// Device/Application/UPM03/UPMRacing_14E_StateMachine_Antigua
FUNCTION_BLOCK UPMRacing_14E_StateMachine_Antigua
VAR_INPUT
	ssMethodType: SINT;
	AMK_bSystemReady1: BOOL;
	AMK_bError1: BOOL;
	AMK_bWarn1: BOOL;
	AMK_bQuitDcOn1: BOOL;
	AMK_bQuitInverterOn1: BOOL;
	AMK_bDerating1: BOOL;
	AMK_ActualVelocity1: INT;
	AMK_TorqueCurrent1: INT;
	AMK_MagnetizingCurrent1: INT;
	AMK_TempMotor1: INT;
	AMK_TempInverter1: INT;
	AMK_ErrorInfo1: UINT;
	AMK_TempIGBT1: INT;
	AMK_bSystemReady2: BOOL;
	AMK_bError2: BOOL;
	AMK_bWarn2: BOOL;
	AMK_bQuitDcOn2: BOOL;
	AMK_bQuitInverterOn2: BOOL;
	AMK_bDerating2: BOOL;
	AMK_ActualVelocity2: INT;
	AMK_TorqueCurrent2: INT;
	AMK_MagnetizingCurrent2: INT;
	AMK_TempMotor2: INT;
	AMK_TempInverter2: INT;
	AMK_ErrorInfo2: UINT;
	AMK_TempIGBT2: INT;
	AMK_bSystemReady3: BOOL;
	AMK_bError3: BOOL;
	AMK_bWarn3: BOOL;
	AMK_bQuitDcOn3: BOOL;
	AMK_bQuitInverterOn3: BOOL;
	AMK_bDerating3: BOOL;
	AMK_ActualVelocity3: INT;
	AMK_TorqueCurrent3: INT;
	AMK_MagnetizingCurrent3: INT;
	AMK_TempMotor3: INT;
	AMK_TempInverter3: INT;
	AMK_ErrorInfo3: UINT;
	AMK_TempIGBT3: INT;
	AMK_bSystemReady4: BOOL;
	AMK_bError4: BOOL;
	AMK_bWarn4: BOOL;
	AMK_bQuitDcOn4: BOOL;
	AMK_bQuitInverterOn4: BOOL;
	AMK_bDerating4: BOOL;
	AMK_ActualVelocity4: INT;
	AMK_TorqueCurrent4: INT;
	AMK_MagnetizingCurrent4: INT;
	AMK_TempMotor4: INT;
	AMK_TempInverter4: INT;
	AMK_ErrorInfo4: UINT;
	AMK_TempIGBT4: INT;
	AccPedal_1: UINT;
	Wake_Up: UINT;
	AMK_bDcOn1_check: BOOL;
	AMK_bDcOn3_check: BOOL;
	AMK_bDcOn2_check: BOOL;
	AMK_bDcOn4_check: BOOL;
	AMK_bInverterOn1_check: BOOL;
	AMK_bInverterOn2_check: BOOL;
	AMK_bInverterOn3_check: BOOL;
	AMK_bInverterOn4_check: BOOL;
	Reset_Button: UINT;
	AccPedal_2: UINT;
	Brake_Pedal: UINT;
	Drive_Button: UINT;
	Speed: REAL;
	Shutdown_Circuit: UINT;
	BMS_Voltage: INT;
	Steering_Wheel_Angle: REAL;
	Yaw_Rate_AIM: INT;
END_VAR
VAR_OUTPUT
	AMK_bInverterOn1: BOOL;
	AMK_bDcOn1: BOOL;
	AMK_bEnable1: BOOL;
	AMK_bErrorReset1: BOOL;
	AMK_TargetVelocity1: INT;
	AMK_TorqueLimitPositiv1: INT;
	AMK_TorqueLimitNegativ1: INT;
	AMK_bInverterOn2: BOOL;
	AMK_bDcOn2: BOOL;
	AMK_bEnable2: BOOL;
	AMK_bErrorReset2: BOOL;
	AMK_TargetVelocity2: INT;
	AMK_TorqueLimitPositiv2: INT;
	AMK_TorqueLimitNegativ2: INT;
	AMK_bInverterOn3: BOOL;
	AMK_bDcOn3: BOOL;
	AMK_bEnable3: BOOL;
	AMK_bErrorReset3: BOOL;
	AMK_TargetVelocity3: INT;
	AMK_TorqueLimitPositiv3: INT;
	AMK_TorqueLimitNegativ3: INT;
	AMK_bInverterOn4: BOOL;
	AMK_bDcOn4: BOOL;
	AMK_bEnable4: BOOL;
	AMK_bErrorReset4: BOOL;
	AMK_TargetVelocity4: INT;
	AMK_TorqueLimitPositiv4: INT;
	AMK_TorqueLimitNegativ4: INT;
	Brake_Light: BOOL;
	Pre_Charge: BOOL;
	Estado: USINT;
	Inverter_Error: BOOL;
	Inverter_Warning: BOOL;
	Info_Inverter_Error: UINT;
	Estado_Error: USINT;
	Fan_Right: BOOL;
	Fan_Left: BOOL;
	RTDS_Sound: BOOL;
	AIM_TempInverter1: USINT;
	AIM_TempInverter2: USINT;
	AIM_TempInverter3: USINT;
	AIM_TempInverter4: USINT;
	AIM_TempMotor1: USINT;
	AIM_TempMotor2: USINT;
	AIM_TempMotor3: USINT;
	AIM_TempMotor4: USINT;
	Cooling_Pumps_On: BOOL;
	AIM_TorqueCurrent1: INT;
	AIM_MagnetizingCurrent1: INT;
	AIM_MagnetizingCurrent2: INT;
	AIM_MagnetizingCurrent3: INT;
	AIM_MagnetizingCurrent4: INT;
	AIM_TargetVelocity1: INT;
	AIM_TargetVelocity2: INT;
	AIM_TargetVelocity3: INT;
	AIM_TargetVelocity4: INT;
	AIM_bDerating1: BOOL;
	AIM_bDerating2: BOOL;
	AIM_bDerating3: BOOL;
	AIM_bDerating4: BOOL;
	AIM_TorqueLimitPositiv1: INT;
	AIM_TorqueLimitPositiv2: INT;
	AIM_TorqueLimitPositiv3: INT;
	AIM_TorqueLimitPositiv4: INT;
	AIM_TorqueCurrent2: INT;
	AIM_TorqueCurrent3: INT;
	AIM_TorqueCurrent4: INT;
	AIM_ActualVelocity1: INT;
	AIM_ActualVelocity2: INT;
	AIM_ActualVelocity3: INT;
	AIM_ActualVelocity4: INT;
	AIM_TempIGBT1: USINT;
	AIM_TempIGBT2: USINT;
	AIM_TempIGBT3: USINT;
	AIM_TempIGBT4: USINT;
	Throttle: REAL;
	Speed_RPM: INT;
	AIM_ErrorInfo1: UINT;
	AIM_ErrorInfo2: UINT;
	AIM_ErrorInfo3: UINT;
	AIM_ErrorInfo4: UINT;
	AIM_bError1: BOOL;
	AIM_bError2: BOOL;
	AIM_bError3: BOOL;
	AIM_bError4: BOOL;
END_VAR
VAR
	Inv_Lower_Temp: INT;
	Motor_Lower_Temp: INT;
	Braking_OffSet: UINT;
	Compare_d: BOOL;
	OutportBufferFory4: INT;
	OutportBufferFory3: INT;
	OutportBufferFory2: INT;
	x_l: INT;
	AMK_bError4_g: BOOL;
	AMK_bError3_n: BOOL;
	AMK_bError2_e: BOOL;
	AMK_bError1_k: BOOL;
	AMK_ErrorInfo4_oa: UINT;
	AMK_ErrorInfo3_p: UINT;
	AMK_ErrorInfo2_a: UINT;
	AMK_ErrorInfo1_h: UINT;
	AMK_MagnetizingCurrent4_m: INT;
	AMK_MagnetizingCurrent3_f: INT;
	AMK_MagnetizingCurrent2_a: INT;
	AMK_MagnetizingCurrent1_j: INT;
	AMK_ActualVelocity4_c: INT;
	AMK_ActualVelocity3_i: INT;
	AMK_ActualVelocity2_e: INT;
	AMK_ActualVelocity1_l: INT;
	AMK_TorqueLimitPositiv4_l: INT;
	AMK_TorqueLimitPositiv3_m: INT;
	AMK_TorqueLimitPositiv2_o: INT;
	AMK_TorqueLimitPositiv1_e: INT;
	AMK_TargetVelocity4_p: INT;
	AMK_TargetVelocity3_h: INT;
	AMK_TargetVelocity2_c: INT;
	AMK_TargetVelocity1_gb: INT;
	AMK_TorqueCurrent4_b: INT;
	AMK_TorqueCurrent3_p: INT;
	AMK_TorqueCurrent2_b: INT;
	AMK_TorqueCurrent1_m: INT;
	AMK_bDerating4_p: BOOL;
	AMK_bDerating3_g: BOOL;
	AMK_bDerating2_p: BOOL;
	AMK_bDerating1_h: BOOL;
	DataTypeConversion3_o: USINT;
	DataTypeConversion1_n: USINT;
	DataTypeConversion2_m: USINT;
	DataTypeConversion_b: USINT;
	DataTypeConversion3_p: USINT;
	DataTypeConversion1_g: USINT;
	DataTypeConversion2_e: USINT;
	DataTypeConversion_e: USINT;
	DataTypeConversion3_e: USINT;
	DataTypeConversion1_c: USINT;
	DataTypeConversion2_f: USINT;
	DataTypeConversion_h: USINT;
	b_Add: UINT;
	OutportBufferForAMK_bErrorReset4: BOOL;
	OutportBufferForAMK_bErrorReset3: BOOL;
	OutportBufferForAMK_bErrorReset2: BOOL;
	Compare: BOOL;
	LogicalOperator1: BOOL;
	LogicalOperator: BOOL;
	Saturation: REAL;
	OutportBufferForAMK_TargetVelocity4: INT;
	OutportBufferForAMK_TargetVelocity3: INT;
	OutportBufferForAMK_TargetVelocity2: INT;
	DataTypeConversion3: INT;
	OutportBufferForAMK_TorqueLimitNegativ4: INT;
	OutportBufferForAMK_TorqueLimitNegativ3: INT;
	OutportBufferForAMK_TorqueLimitNegativ2: INT;
	DataTypeConversion6: INT;
	DataTypeConversion: INT;
	DataTypeConversion5: INT;
	DataTypeConversion4: INT;
	DataTypeConversion2: INT;
	DataTypeConversion1: INT;
	is_active_c3_UPMRacing_14E_StateMachine: USINT;
	is_CAR: USINT;
	is_SHUTDOWN_SEQUENCE: USINT;
	temporalCounter_i1: PLC_CODER_TIMER;
	Cooling_Enable: BOOL;
	x: INT;
	is_IDLE: USINT;
	is_DRIVE: USINT;
	BMS_Voltage_Min: INT;
	b_AccPedal_2: UINT;
	b_AccPedal_1: UINT;
	b_Yaw_Rate_AIM: INT;
	b_Steering_Wheel_Angle: REAL;
	Throttle_a: REAL;
	b_AMK_ActualVelocity4: INT;
	b_AMK_ActualVelocity3: INT;
	b_AMK_ActualVelocity2: INT;
	b_AMK_ActualVelocity1: INT;
	is_POWER_MOTOR_ON: USINT;
	is_ERROR_INVERTER: USINT;
	b_AMK_bWarn4: BOOL;
	b_AMK_bWarn3: BOOL;
	b_AMK_bWarn2: BOOL;
	b_AMK_bWarn1: BOOL;
	b_AMK_bError4: BOOL;
	b_AMK_bError3: BOOL;
	b_AMK_bError2: BOOL;
	b_AMK_bError1: BOOL;
	AMK_bError4_a: BOOL;
	AMK_bError3_d: BOOL;
	AMK_bError2_h: BOOL;
	AMK_bError1_b: BOOL;
	b_AMK_ErrorInfo4: UINT;
	b_AMK_ErrorInfo3: UINT;
	b_AMK_ErrorInfo2: UINT;
	b_AMK_ErrorInfo1: UINT;
	is_BRAKE_LIGHT: USINT;
	is_COOLING_RIGHT: USINT;
	Fan_Upper_Speed: UINT;
	Motor_Upper_Temp: INT;
	Fan_Lower_Speed: UINT;
	is_COOLING_LEFT: USINT;
	b_AMK_TempInverter4: INT;
	b_AMK_TempInverter3: INT;
	b_AMK_TempInverter2: INT;
	b_AMK_TempInverter1: INT;
	b_AMK_TempMotor4: INT;
	b_AMK_TempMotor3: INT;
	b_AMK_TempMotor2: INT;
	b_AMK_TempMotor1: INT;
	b_AMK_TempIGBT4: INT;
	b_AMK_TempIGBT3: INT;
	b_AMK_TempIGBT2: INT;
	b_AMK_TempIGBT1: INT;
	b_AMK_bDerating4: BOOL;
	b_AMK_bDerating3: BOOL;
	b_AMK_bDerating2: BOOL;
	b_AMK_bDerating1: BOOL;
	b_AMK_TorqueCurrent4: INT;
	b_AMK_TorqueCurrent3: INT;
	b_AMK_TorqueCurrent2: INT;
	b_AMK_TorqueCurrent1: INT;
	AMK_TargetVelocity4_b: INT;
	AMK_TargetVelocity3_m: INT;
	AMK_TargetVelocity2_m: INT;
	AMK_TargetVelocity1_g: INT;
	AMK_TorqueLimitPositiv4_h: INT;
	AMK_TorqueLimitPositiv3_i: INT;
	AMK_TorqueLimitPositiv2_l: INT;
	AMK_TorqueLimitPositiv1_c: INT;
	AMK_ActualVelocity4_k: INT;
	AMK_ActualVelocity3_f: INT;
	AMK_ActualVelocity2_n: INT;
	AMK_ActualVelocity1_b: INT;
	b_AMK_MagnetizingCurrent4: INT;
	b_AMK_MagnetizingCurrent3: INT;
	b_AMK_MagnetizingCurrent2: INT;
	b_AMK_MagnetizingCurrent1: INT;
	AMK_bError4_p: BOOL;
	AMK_bError3_p: BOOL;
	AMK_bError2_g: BOOL;
	AMK_bError1_d: BOOL;
	AMK_ErrorInfo4_o: UINT;
	AMK_ErrorInfo3_l: UINT;
	AMK_ErrorInfo2_f: UINT;
	AMK_ErrorInfo1_n: UINT;
	Inv_Upper_Temp: INT;
	i0_b_Constant: b_Constant;
	i0_Throttle_Control: Throttle_Control;
	i0_Yaw_Control: Yaw_Control;
	i0_Error_Control: Error_Control;
	i0_Error_RESET: Error_RESET;
	i0_Error_Info: Error_Info;
	i0_Temp_Inverter: Temp_Inverter;
	i0_Temp_Motor: Temp_Motor;
	i0_Temp_IGBT: Temp_IGBT;
	i0_Derating: Derating;
	i0_TorqueCurrent: TorqueCurrent;
	i0_TargetVelocity: TargetVelocity;
	i0_TorqueLimitPositiv: TorqueLimitPositiv;
	i0_ActualVelocity: ActualVelocity;
	i0_MagnetizingCurrent: MagnetizingCurrent;
	i0_ErrorInfo: ErrorInfo;
	sf_internal_predicateOutput: BOOL;
	tmp: UINT;
	temp1: UINT;
	temp2: UINT;
	temp3: USINT;
	temp4: USINT;
	temp5: USINT;
	temp6: USINT;
	temp7: UINT;
	temp8: BOOL;
	temp9: BOOL;
	temp10: BOOL;
	temp11: REAL;
	temp12: INT;
	temp13: INT;
	temp14: INT;
	temp15: INT;
	temp16: INT;
	temp17: INT;
	temp18: INT;
	temp19: INT;
	temp20: INT;
	temp21: INT;
	temp22: INT;
	temp23: INT;
	temp24: INT;
	
	//Llamadas a las funciones de CAN (Copiar)
	
	CAN_RX_V_1_2:CAN_RX_V_1_2;
	CAN_RX_Inverters:CAN_RX_Inverters;
	
	CAN_TX_V_1_4:CAN_TX_V_1_4;
	CAN_TX_Inverters:CAN_TX_Inverters;
	
END_VAR


CAN_RX_V_1_2( 
	    		
		(*DATA LOGGER*) (*
			DL_Msg_Cntr_CAN => DL_Msg_Cntr,
			DL_Status_CAN => DL_Status,
			DL_Power_CAN => DL_Power,
			DL_Voltage_CAN => DL_Voltage,
			DL_Current_CAN => DL_Current,
		(*FIN DATA LOGGER*) *)
		
		(*BMS*)
			BatVoltage_MSB_CAN => BMS_Voltage,
		(*__*)
		
		(*AIM RX*) 
			Speed_CAN => Speed,
			//AIM_Long_Acc_CAN => Long_Acc,
			//AIM_Lat_Acc_CAN => Lat_Acc,
			Yaw_Rate_AIM_CAN => Yaw_Rate_AIM, 
			
			Steering_Wheel_Angle_CAN => Steering_Wheel_Angle,
		(*__*)
		
			); 	
(*_________*)		
		
CAN_RX_Inverters( 
	
		(*INVERTERS*)
		AMK_bSystemReady1_CAN=>AMK_bSystemReady1,
		AMK_bError1_CAN=>AMK_bError1,
		AMK_bWarn1_CAN=>AMK_bWarn1,
		AMK_bQuitDcOn1_CAN=>AMK_bQuitDcOn1,
		AMK_bDcOn1_check_CAN=>AMK_bDcOn1_check,
		AMK_bQuitInverterOn1_CAN=>AMK_bQuitInverterOn1,
		AMK_bInverterOn1_check_CAN=>AMK_bInverterOn1_check,
		AMK_bDerating1_CAN=>AMK_bDerating1,
		AMK_ActualVelocity1_CAN=>AMK_ActualVelocity1,
		AMK_TorqueCurrent1_CAN=>AMK_TorqueCurrent1,
		AMK_MagnetizingCurrent1_CAN=>AMK_MagnetizingCurrent1,
		AMK_TempMotor1_CAN=>AMK_TempMotor1,
		AMK_TempInverter1_CAN=>AMK_TempInverter1,
		AMK_ErrorInfo1_CAN=>AMK_ErrorInfo1,
		AMK_TempIGBT1_CAN=>AMK_TempIGBT1,
		
		
		AMK_bSystemReady2_CAN=>AMK_bSystemReady2,
		AMK_bError2_CAN=>AMK_bError2,
		AMK_bWarn2_CAN=>AMK_bWarn2,
		AMK_bQuitDcOn2_CAN=>AMK_bQuitDcOn2,
		AMK_bDcOn2_check_CAN=>AMK_bDcOn2_check,
		AMK_bQuitInverterOn2_CAN=>AMK_bQuitInverterOn2,
		AMK_bInverterOn2_check_CAN=>AMK_bInverterOn2_check,
		AMK_bDerating2_CAN=>AMK_bDerating2,
		AMK_ActualVelocity2_CAN=>AMK_ActualVelocity2,
		AMK_TorqueCurrent2_CAN=>AMK_TorqueCurrent2,
		AMK_MagnetizingCurrent2_CAN=>AMK_MagnetizingCurrent2,
		AMK_TempMotor2_CAN=>AMK_TempMotor2,
		AMK_TempInverter2_CAN=>AMK_TempInverter2,
		AMK_ErrorInfo2_CAN=>AMK_ErrorInfo2,
		AMK_TempIGBT2_CAN=>AMK_TempIGBT2,
		
		
		AMK_bSystemReady3_CAN=>AMK_bSystemReady3,
		AMK_bError3_CAN=>AMK_bError3,
		AMK_bWarn3_CAN=>AMK_bWarn3,
		AMK_bQuitDcOn3_CAN=>AMK_bQuitDcOn3,
		AMK_bDcOn3_check_CAN=>AMK_bDcOn3_check,
		AMK_bQuitInverterOn3_CAN=>AMK_bQuitInverterOn3,
		AMK_bInverterOn3_check_CAN=>AMK_bInverterOn3_check,
		AMK_bDerating3_CAN=>AMK_bDerating3,
		AMK_ActualVelocity3_CAN=>AMK_ActualVelocity3,
		AMK_TorqueCurrent3_CAN=>AMK_TorqueCurrent3,
		AMK_MagnetizingCurrent3_CAN=>AMK_MagnetizingCurrent3,
		AMK_TempMotor3_CAN=>AMK_TempMotor3,
		AMK_TempInverter3_CAN=>AMK_TempInverter3,
		AMK_ErrorInfo3_CAN=>AMK_ErrorInfo3,
		AMK_TempIGBT3_CAN=>AMK_TempIGBT3,
		
		
		AMK_bSystemReady4_CAN=>AMK_bSystemReady4,
		AMK_bError4_CAN=>AMK_bError4,
		AMK_bWarn4_CAN=>AMK_bWarn4,
		AMK_bQuitDcOn4_CAN=>AMK_bQuitDcOn4,
		AMK_bDcOn4_check_CAN=>AMK_bDcOn4_check,
		AMK_bQuitInverterOn4_CAN=>AMK_bQuitInverterOn4,
		AMK_bInverterOn4_check_CAN=>AMK_bInverterOn4_check,
		AMK_bDerating4_CAN=>AMK_bDerating4,
		AMK_ActualVelocity4_CAN=>AMK_ActualVelocity4,
		AMK_TorqueCurrent4_CAN=>AMK_TorqueCurrent4,
		AMK_MagnetizingCurrent4_CAN=>AMK_MagnetizingCurrent4,
		AMK_TempMotor4_CAN=>AMK_TempMotor4,
		AMK_TempInverter4_CAN=>AMK_TempInverter4,
		AMK_ErrorInfo4_CAN=>AMK_ErrorInfo4,
		AMK_TempIGBT4_CAN=>AMK_TempIGBT4
		
		);

(*___________________*)

CASE ssMethodType OF
    SS_INITIALIZE: 
        (* SystemInitialize for Chart: '<Root>/UPMRacing_14E_StateMachine' incorporates:
         *  Outport: '<Root>/AIM_ErrorInfo1'
         *  Outport: '<Root>/AIM_ErrorInfo2'
         *  Outport: '<Root>/AIM_ErrorInfo3'
         *  Outport: '<Root>/AIM_ErrorInfo4'
         *  Outport: '<Root>/AIM_TargetVelocity1'
         *  Outport: '<Root>/AIM_TargetVelocity2'
         *  Outport: '<Root>/AIM_TargetVelocity3'
         *  Outport: '<Root>/AIM_TargetVelocity4'
         *  Outport: '<Root>/AIM_TorqueLimitPositiv1'
         *  Outport: '<Root>/AIM_TorqueLimitPositiv2'
         *  Outport: '<Root>/AIM_TorqueLimitPositiv3'
         *  Outport: '<Root>/AIM_TorqueLimitPositiv4'
         *  Outport: '<Root>/AIM_bError1'
         *  Outport: '<Root>/AIM_bError2'
         *  Outport: '<Root>/AIM_bError3'
         *  Outport: '<Root>/AIM_bError4'
         *  Outport: '<Root>/AMK_TargetVelocity1'
         *  Outport: '<Root>/AMK_TargetVelocity2'
         *  Outport: '<Root>/AMK_TargetVelocity3'
         *  Outport: '<Root>/AMK_TargetVelocity4'
         *  Outport: '<Root>/AMK_TorqueLimitNegativ1'
         *  Outport: '<Root>/AMK_TorqueLimitNegativ2'
         *  Outport: '<Root>/AMK_TorqueLimitNegativ3'
         *  Outport: '<Root>/AMK_TorqueLimitNegativ4'
         *  Outport: '<Root>/AMK_TorqueLimitPositiv1'
         *  Outport: '<Root>/AMK_TorqueLimitPositiv2'
         *  Outport: '<Root>/AMK_TorqueLimitPositiv3'
         *  Outport: '<Root>/AMK_TorqueLimitPositiv4'
         *  Outport: '<Root>/AMK_bDcOn1'
         *  Outport: '<Root>/AMK_bDcOn2'
         *  Outport: '<Root>/AMK_bDcOn3'
         *  Outport: '<Root>/AMK_bDcOn4'
         *  Outport: '<Root>/AMK_bEnable1'
         *  Outport: '<Root>/AMK_bEnable2'
         *  Outport: '<Root>/AMK_bEnable3'
         *  Outport: '<Root>/AMK_bEnable4'
         *  Outport: '<Root>/AMK_bErrorReset1'
         *  Outport: '<Root>/AMK_bErrorReset2'
         *  Outport: '<Root>/AMK_bErrorReset3'
         *  Outport: '<Root>/AMK_bErrorReset4'
         *  Outport: '<Root>/AMK_bInverterOn1'
         *  Outport: '<Root>/AMK_bInverterOn2'
         *  Outport: '<Root>/AMK_bInverterOn3'
         *  Outport: '<Root>/AMK_bInverterOn4'
         *  Outport: '<Root>/Fan_Left'
         *  Outport: '<Root>/Fan_Right'
         *  Outport: '<Root>/RTDS_Sound'
         *  Outport: '<Root>/Speed_RPM' *)
        is_BRAKE_LIGHT := UPMRacing_14E_StateMachine_IN_NO_ACTIVE_CHILD;
        is_CAR := UPMRacing_14E_StateMachine_IN_NO_ACTIVE_CHILD;
        is_DRIVE := UPMRacing_14E_StateMachine_IN_NO_ACTIVE_CHILD;
        temporalCounter_i1(timerAction := 1, maxTime := 0);
        is_IDLE := UPMRacing_14E_StateMachine_IN_NO_ACTIVE_CHILD;
        is_POWER_MOTOR_ON := UPMRacing_14E_StateMachine_IN_NO_ACTIVE_CHILD;
        temporalCounter_i1(timerAction := 1, maxTime := 0);
        is_SHUTDOWN_SEQUENCE := UPMRacing_14E_StateMachine_IN_NO_ACTIVE_CHILD;
        temporalCounter_i1(timerAction := 1, maxTime := 0);
        is_COOLING_LEFT := UPMRacing_14E_StateMachine_IN_NO_ACTIVE_CHILD;
        is_COOLING_RIGHT := UPMRacing_14E_StateMachine_IN_NO_ACTIVE_CHILD;
        is_ERROR_INVERTER := UPMRacing_14E_StateMachine_IN_NO_ACTIVE_CHILD;
        is_active_c3_UPMRacing_14E_StateMachine := 0;
        Braking_OffSet := 3850;
        Motor_Upper_Temp := 700;
        Motor_Lower_Temp := 500;
        Fan_Upper_Speed := 350;
        Fan_Lower_Speed := 350;
        Inv_Lower_Temp := 250;
        Inv_Upper_Temp := 300;
        Cooling_Enable := FALSE;
        BMS_Voltage_Min := 306;
        AMK_bInverterOn1 := FALSE;
        AMK_bDcOn1 := FALSE;
        AMK_bEnable1 := FALSE;
        AMK_bErrorReset1 := FALSE;
        AMK_TargetVelocity1 := 0;
        AMK_TorqueLimitPositiv1 := 0;
        AMK_TorqueLimitNegativ1 := 0;
        AMK_bInverterOn2 := FALSE;
        AMK_bDcOn2 := FALSE;
        AMK_bEnable2 := FALSE;
        AMK_bErrorReset2 := FALSE;
        AMK_TargetVelocity2 := 0;
        AMK_TorqueLimitPositiv2 := 0;
        AMK_TorqueLimitNegativ2 := 0;
        AMK_bInverterOn3 := FALSE;
        AMK_bDcOn3 := FALSE;
        AMK_bEnable3 := FALSE;
        AMK_bErrorReset3 := FALSE;
        AMK_TargetVelocity3 := 0;
        AMK_TorqueLimitPositiv3 := 0;
        AMK_TorqueLimitNegativ3 := 0;
        AMK_bInverterOn4 := FALSE;
        AMK_bDcOn4 := FALSE;
        AMK_bEnable4 := FALSE;
        AMK_bErrorReset4 := FALSE;
        AMK_TargetVelocity4 := 0;
        AMK_TorqueLimitPositiv4 := 0;
        AMK_TorqueLimitNegativ4 := 0;
        Fan_Right := FALSE;
        Fan_Left := FALSE;
        RTDS_Sound := FALSE;
        AIM_TargetVelocity1 := 0;
        AIM_TargetVelocity2 := 0;
        AIM_TargetVelocity3 := 0;
        AIM_TargetVelocity4 := 0;
        AIM_TorqueLimitPositiv1 := 0;
        AIM_TorqueLimitPositiv2 := 0;
        AIM_TorqueLimitPositiv3 := 0;
        AIM_TorqueLimitPositiv4 := 0;
        Speed_RPM := 0;
        AIM_ErrorInfo1 := 0;
        AIM_ErrorInfo2 := 0;
        AIM_ErrorInfo3 := 0;
        AIM_ErrorInfo4 := 0;
        AIM_bError1 := FALSE;
        AIM_bError2 := FALSE;
        AIM_bError3 := FALSE;
        AIM_bError4 := FALSE;
        i0_Yaw_Control(ssMethodType := SS_INITIALIZE, AMK_ActualVelocity1 := b_AMK_ActualVelocity1, AMK_ActualVelocity2 := b_AMK_ActualVelocity2, AMK_ActualVelocity3 := b_AMK_ActualVelocity3, AMK_ActualVelocity4 := b_AMK_ActualVelocity4, Throttle := Throttle_a, Steering_Wheel_Angle := b_Steering_Wheel_Angle, Yaw_Rate_AIM := b_Yaw_Rate_AIM);
        OutportBufferForAMK_TargetVelocity4 := temp24;
        OutportBufferForAMK_TargetVelocity3 := temp23;
        OutportBufferForAMK_TargetVelocity2 := temp22;
        DataTypeConversion3 := temp21;
        OutportBufferForAMK_TorqueLimitNegativ4 := temp20;
        OutportBufferForAMK_TorqueLimitNegativ3 := temp19;
        OutportBufferForAMK_TorqueLimitNegativ2 := temp18;
        DataTypeConversion6 := temp17;
        DataTypeConversion := temp16;
        DataTypeConversion5 := temp15;
        DataTypeConversion4 := temp14;
        DataTypeConversion2 := temp13;
        DataTypeConversion1 := temp12;
        i0_b_Constant(ssMethodType := SS_INITIALIZE, x := x);
        OutportBufferFory4 := temp15;
        OutportBufferFory3 := temp14;
        OutportBufferFory2 := temp13;
        x_l := temp12;
        i0_Throttle_Control(ssMethodType := SS_INITIALIZE, AccPedal_1 := b_AccPedal_1, AccPedal_2 := b_AccPedal_2,  Brake_Light2 := Brake_Pedal);
        Compare_d := sf_internal_predicateOutput;
        Saturation := temp11;
        i0_Error_Control(ssMethodType := SS_INITIALIZE, AMK_bError1 := b_AMK_bError1, AMK_bError2 := b_AMK_bError2, AMK_bError3 := b_AMK_bError3, AMK_bError4 := b_AMK_bError4, AMK_bWarn1 := b_AMK_bWarn1, AMK_bWarn2 := b_AMK_bWarn2, AMK_bWarn3 := b_AMK_bWarn3, AMK_bWarn4 := b_AMK_bWarn4);
        LogicalOperator1 := temp10;
        LogicalOperator := sf_internal_predicateOutput;
        i0_Error_RESET(ssMethodType := SS_INITIALIZE);
        OutportBufferForAMK_bErrorReset4 := temp9;
        OutportBufferForAMK_bErrorReset3 := temp8;
        OutportBufferForAMK_bErrorReset2 := temp10;
        Compare := sf_internal_predicateOutput;
        i0_Error_Info(ssMethodType := SS_INITIALIZE, AMK_ErrorInfo1 := b_AMK_ErrorInfo1, AMK_ErrorInfo2 := b_AMK_ErrorInfo2, AMK_ErrorInfo3 := b_AMK_ErrorInfo3, AMK_ErrorInfo4 := b_AMK_ErrorInfo4, AMK_bError1 := AMK_bError1_b, AMK_bError2 := AMK_bError2_h, AMK_bError3 := AMK_bError3_d, AMK_bError4 := AMK_bError4_a);
        b_Add := temp7;
        i0_Temp_Inverter(ssMethodType := SS_INITIALIZE, AMK_TempInverter1 := b_AMK_TempInverter1, AMK_TempInverter2 := b_AMK_TempInverter2, AMK_TempInverter3 := b_AMK_TempInverter3, AMK_TempInverter4 := b_AMK_TempInverter4);
        DataTypeConversion3_e := temp6;
        DataTypeConversion1_c := temp5;
        DataTypeConversion2_f := temp4;
        DataTypeConversion_h := temp3;
        i0_Temp_Motor(ssMethodType := SS_INITIALIZE, AMK_TempMotor1 := b_AMK_TempMotor1, AMK_TempMotor2 := b_AMK_TempMotor2, AMK_TempMotor3 := b_AMK_TempMotor3, AMK_TempMotor4 := b_AMK_TempMotor4);
        DataTypeConversion3_p := temp6;
        DataTypeConversion1_g := temp5;
        DataTypeConversion2_e := temp4;
        DataTypeConversion_e := temp3;
        i0_Temp_IGBT(ssMethodType := SS_INITIALIZE, AMK_TempIGBT1 := b_AMK_TempIGBT1, AMK_TempIGBT2 := b_AMK_TempIGBT2, AMK_TempIGBT3 := b_AMK_TempIGBT3, AMK_TempIGBT4 := b_AMK_TempIGBT4);
        DataTypeConversion3_o := temp6;
        DataTypeConversion1_n := temp5;
        DataTypeConversion2_m := temp4;
        DataTypeConversion_b := temp3;
        i0_Derating(ssMethodType := SS_INITIALIZE, AMK_bDerating1 := b_AMK_bDerating1, AMK_bDerating2 := b_AMK_bDerating2, AMK_bDerating3 := b_AMK_bDerating3, AMK_bDerating4 := b_AMK_bDerating4);
        AMK_bDerating4_p := temp9;
        AMK_bDerating3_g := temp8;
        AMK_bDerating2_p := temp10;
        AMK_bDerating1_h := sf_internal_predicateOutput;
        i0_MagnetizingCurrent(ssMethodType := SS_INITIALIZE, AMK_MagnetizingCurrent1 := b_AMK_MagnetizingCurrent1, AMK_MagnetizingCurrent2 := b_AMK_MagnetizingCurrent2, AMK_MagnetizingCurrent3 := b_AMK_MagnetizingCurrent3, AMK_MagnetizingCurrent4 := b_AMK_MagnetizingCurrent4);
        AMK_MagnetizingCurrent4_m := temp15;
        AMK_MagnetizingCurrent3_f := temp14;
        AMK_MagnetizingCurrent2_a := temp13;
        AMK_MagnetizingCurrent1_j := temp12;
        i0_TorqueCurrent(ssMethodType := SS_INITIALIZE, AMK_TorqueCurrent1 := b_AMK_TorqueCurrent1, AMK_TorqueCurrent2 := b_AMK_TorqueCurrent2, AMK_TorqueCurrent3 := b_AMK_TorqueCurrent3, AMK_TorqueCurrent4 := b_AMK_TorqueCurrent4);
        AMK_TorqueCurrent4_b := temp15;
        AMK_TorqueCurrent3_p := temp14;
        AMK_TorqueCurrent2_b := temp13;
        AMK_TorqueCurrent1_m := temp12;
        i0_TargetVelocity(ssMethodType := SS_INITIALIZE, AMK_TargetVelocity1 := AMK_TargetVelocity1_g, AMK_TargetVelocity2 := AMK_TargetVelocity2_m, AMK_TargetVelocity3 := AMK_TargetVelocity3_m, AMK_TargetVelocity4 := AMK_TargetVelocity4_b);
        AMK_TargetVelocity4_p := temp15;
        AMK_TargetVelocity3_h := temp14;
        AMK_TargetVelocity2_c := temp13;
        AMK_TargetVelocity1_gb := temp12;
        i0_TorqueLimitPositiv(ssMethodType := SS_INITIALIZE, AMK_TorqueLimitPositiv1 := AMK_TorqueLimitPositiv1_c, AMK_TorqueLimitPositiv2 := AMK_TorqueLimitPositiv2_l, AMK_TorqueLimitPositiv3 := AMK_TorqueLimitPositiv3_i, AMK_TorqueLimitPositiv4 := AMK_TorqueLimitPositiv4_h);
        AMK_TorqueLimitPositiv4_l := temp15;
        AMK_TorqueLimitPositiv3_m := temp14;
        AMK_TorqueLimitPositiv2_o := temp13;
        AMK_TorqueLimitPositiv1_e := temp12;
        i0_ActualVelocity(ssMethodType := SS_INITIALIZE, AMK_ActualVelocity1 := AMK_ActualVelocity1_b, AMK_ActualVelocity2 := AMK_ActualVelocity2_n, AMK_ActualVelocity3 := AMK_ActualVelocity3_f, AMK_ActualVelocity4 := AMK_ActualVelocity4_k);
        AMK_ActualVelocity4_c := temp15;
        AMK_ActualVelocity3_i := temp14;
        AMK_ActualVelocity2_e := temp13;
        AMK_ActualVelocity1_l := temp12;
        i0_ErrorInfo(ssMethodType := SS_INITIALIZE, AMK_ErrorInfo1 := AMK_ErrorInfo1_n, AMK_ErrorInfo2 := AMK_ErrorInfo2_f, AMK_ErrorInfo3 := AMK_ErrorInfo3_l, AMK_ErrorInfo4 := AMK_ErrorInfo4_o, AMK_bError1 := AMK_bError1_d, AMK_bError2 := AMK_bError2_g, AMK_bError3 := AMK_bError3_p, AMK_bError4 := AMK_bError4_p);
        AMK_bError4_g := temp9;
        AMK_bError3_n := temp8;
        AMK_bError2_e := temp10;
        AMK_bError1_k := sf_internal_predicateOutput;
        AMK_ErrorInfo4_oa := temp2;
        AMK_ErrorInfo3_p := temp1;
        AMK_ErrorInfo2_a := tmp;
        AMK_ErrorInfo1_h := temp7;
    SS_STEP: 
        (* Chart: '<Root>/UPMRacing_14E_StateMachine' incorporates:
         *  Outport: '<Root>/AIM_ActualVelocity1'
         *  Outport: '<Root>/AIM_ActualVelocity2'
         *  Outport: '<Root>/AIM_ActualVelocity3'
         *  Outport: '<Root>/AIM_ActualVelocity4'
         *  Outport: '<Root>/AIM_ErrorInfo1'
         *  Outport: '<Root>/AIM_ErrorInfo2'
         *  Outport: '<Root>/AIM_ErrorInfo3'
         *  Outport: '<Root>/AIM_ErrorInfo4'
         *  Outport: '<Root>/AIM_MagnetizingCurrent1'
         *  Outport: '<Root>/AIM_MagnetizingCurrent2'
         *  Outport: '<Root>/AIM_MagnetizingCurrent3'
         *  Outport: '<Root>/AIM_MagnetizingCurrent4'
         *  Outport: '<Root>/AIM_TargetVelocity1'
         *  Outport: '<Root>/AIM_TargetVelocity2'
         *  Outport: '<Root>/AIM_TargetVelocity3'
         *  Outport: '<Root>/AIM_TargetVelocity4'
         *  Outport: '<Root>/AIM_TempIGBT1'
         *  Outport: '<Root>/AIM_TempIGBT2'
         *  Outport: '<Root>/AIM_TempIGBT3'
         *  Outport: '<Root>/AIM_TempIGBT4'
         *  Outport: '<Root>/AIM_TempInverter1'
         *  Outport: '<Root>/AIM_TempInverter2'
         *  Outport: '<Root>/AIM_TempInverter3'
         *  Outport: '<Root>/AIM_TempInverter4'
         *  Outport: '<Root>/AIM_TempMotor1'
         *  Outport: '<Root>/AIM_TempMotor2'
         *  Outport: '<Root>/AIM_TempMotor3'
         *  Outport: '<Root>/AIM_TempMotor4'
         *  Outport: '<Root>/AIM_TorqueCurrent1'
         *  Outport: '<Root>/AIM_TorqueCurrent2'
         *  Outport: '<Root>/AIM_TorqueCurrent3'
         *  Outport: '<Root>/AIM_TorqueCurrent4'
         *  Outport: '<Root>/AIM_TorqueLimitPositiv1'
         *  Outport: '<Root>/AIM_TorqueLimitPositiv2'
         *  Outport: '<Root>/AIM_TorqueLimitPositiv3'
         *  Outport: '<Root>/AIM_TorqueLimitPositiv4'
         *  Outport: '<Root>/AIM_bDerating1'
         *  Outport: '<Root>/AIM_bDerating2'
         *  Outport: '<Root>/AIM_bDerating3'
         *  Outport: '<Root>/AIM_bDerating4'
         *  Outport: '<Root>/AIM_bError1'
         *  Outport: '<Root>/AIM_bError2'
         *  Outport: '<Root>/AIM_bError3'
         *  Outport: '<Root>/AIM_bError4'
         *  Outport: '<Root>/AMK_TargetVelocity1'
         *  Outport: '<Root>/AMK_TargetVelocity2'
         *  Outport: '<Root>/AMK_TargetVelocity3'
         *  Outport: '<Root>/AMK_TargetVelocity4'
         *  Outport: '<Root>/AMK_TorqueLimitNegativ1'
         *  Outport: '<Root>/AMK_TorqueLimitNegativ2'
         *  Outport: '<Root>/AMK_TorqueLimitNegativ3'
         *  Outport: '<Root>/AMK_TorqueLimitNegativ4'
         *  Outport: '<Root>/AMK_TorqueLimitPositiv1'
         *  Outport: '<Root>/AMK_TorqueLimitPositiv2'
         *  Outport: '<Root>/AMK_TorqueLimitPositiv3'
         *  Outport: '<Root>/AMK_TorqueLimitPositiv4'
         *  Outport: '<Root>/AMK_bDcOn1'
         *  Outport: '<Root>/AMK_bDcOn2'
         *  Outport: '<Root>/AMK_bDcOn3'
         *  Outport: '<Root>/AMK_bDcOn4'
         *  Outport: '<Root>/AMK_bEnable1'
         *  Outport: '<Root>/AMK_bEnable2'
         *  Outport: '<Root>/AMK_bEnable3'
         *  Outport: '<Root>/AMK_bEnable4'
         *  Outport: '<Root>/AMK_bErrorReset1'
         *  Outport: '<Root>/AMK_bErrorReset2'
         *  Outport: '<Root>/AMK_bErrorReset3'
         *  Outport: '<Root>/AMK_bErrorReset4'
         *  Outport: '<Root>/AMK_bInverterOn1'
         *  Outport: '<Root>/AMK_bInverterOn2'
         *  Outport: '<Root>/AMK_bInverterOn3'
         *  Outport: '<Root>/AMK_bInverterOn4'
         *  Outport: '<Root>/Brake_Light'
         *  Outport: '<Root>/Cooling_Pumps_On'
         *  Outport: '<Root>/Estado'
         *  Outport: '<Root>/Fan_Left'
         *  Outport: '<Root>/Fan_Right'
         *  Outport: '<Root>/Info_Inverter_Error'
         *  Outport: '<Root>/Inverter_Error'
         *  Outport: '<Root>/Inverter_Warning'
         *  Outport: '<Root>/Pre_Charge'
         *  Outport: '<Root>/RTDS_Sound'
         *  Outport: '<Root>/Speed_RPM'
         *  Outport: '<Root>/Throttle' *)
        (* Gateway: UPMRacing_14E_StateMachine *)
        (* During: UPMRacing_14E_StateMachine *)

        IF is_active_c3_UPMRacing_14E_StateMachine = 0 THEN 
            (* Entry: UPMRacing_14E_StateMachine *)
            is_active_c3_UPMRacing_14E_StateMachine := 1;
            (* Entry Internal: UPMRacing_14E_StateMachine *)
            (* Entry Internal 'CAR': '<S1>:380' *)
            (* Transition: '<S1>:138' *)
            is_CAR := UPMRacing_14E_StateMachine_IN_IDLE;
            (* Entry 'IDLE': '<S1>:333' *)
            (* '<S1>:333:3' Cooling_Enable = false; *)
            Cooling_Enable := FALSE;
            (* '<S1>:333:4' [AMK_TargetVelocity1, AMK_TargetVelocity2, AMK_TargetVelocity3, AMK_TargetVelocity4... *)
            (* '<S1>:333:5'      ]=Constant(int16(0)); *)
            (* Simulink Function 'Constant': '<S1>:190' *)
            x := 0;
            i0_b_Constant(ssMethodType := SS_OUTPUT, x := x);
            temp12 := i0_b_Constant.y1;
            temp13 := i0_b_Constant.y2;
            temp14 := i0_b_Constant.y3;
            temp15 := i0_b_Constant.y4;
            OutportBufferFory4 := temp15;
            OutportBufferFory3 := temp14;
            OutportBufferFory2 := temp13;
            x_l := temp12;
            AMK_TargetVelocity1 := x_l;
            AMK_TargetVelocity2 := OutportBufferFory2;
            AMK_TargetVelocity3 := OutportBufferFory3;
            AMK_TargetVelocity4 := OutportBufferFory4;
            (* '<S1>:333:6' [AMK_TorqueLimitPositiv1, AMK_TorqueLimitPositiv2, AMK_TorqueLimitPositiv3,... *)
            (* '<S1>:333:7'      AMK_TorqueLimitPositiv4]=Constant(int16(0)); *)
            (* Simulink Function 'Constant': '<S1>:190' *)
            x := 0;
            i0_b_Constant(ssMethodType := SS_OUTPUT, x := x);
            temp12 := i0_b_Constant.y1;
            temp13 := i0_b_Constant.y2;
            temp14 := i0_b_Constant.y3;
            temp15 := i0_b_Constant.y4;
            OutportBufferFory4 := temp15;
            OutportBufferFory3 := temp14;
            OutportBufferFory2 := temp13;
            x_l := temp12;
            AMK_TorqueLimitPositiv1 := x_l;
            AMK_TorqueLimitPositiv2 := OutportBufferFory2;
            AMK_TorqueLimitPositiv3 := OutportBufferFory3;
            AMK_TorqueLimitPositiv4 := OutportBufferFory4;
            (* '<S1>:333:8' [AMK_TorqueLimitNegativ1, AMK_TorqueLimitNegativ2, AMK_TorqueLimitNegativ3, ... *)
            (* '<S1>:333:9'      AMK_TorqueLimitNegativ4]=Constant(int16(0)); *)
            (* Simulink Function 'Constant': '<S1>:190' *)
            x := 0;
            i0_b_Constant(ssMethodType := SS_OUTPUT, x := x);
            temp12 := i0_b_Constant.y1;
            temp13 := i0_b_Constant.y2;
            temp14 := i0_b_Constant.y3;
            temp15 := i0_b_Constant.y4;
            OutportBufferFory4 := temp15;
            OutportBufferFory3 := temp14;
            OutportBufferFory2 := temp13;
            x_l := temp12;
            AMK_TorqueLimitNegativ1 := x_l;
            AMK_TorqueLimitNegativ2 := OutportBufferFory2;
            AMK_TorqueLimitNegativ3 := OutportBufferFory3;
            AMK_TorqueLimitNegativ4 := OutportBufferFory4;
            (* Entry Internal 'IDLE': '<S1>:333' *)
            (* Transition: '<S1>:335' *)
            is_IDLE := UPMRacing_14E_StateMachine_IN_LVMS_ON;
            (* Entry 'LVMS_ON': '<S1>:334' *)
            (* In this state the ECU is waiting to start the inizialization of the inverters *)
            (* Right now all LV systems are starting to initialize *)
            (* '<S1>:334:4' Estado = 1; *)
            Estado := 1;
            (* Battery relays *)
            (* '<S1>:334:6' Pre_Charge = false; *)
            Pre_Charge := FALSE;
            (* Inverters shutdown *)
            (* '<S1>:334:8' AMK_bInverterOn1=false; *)
            AMK_bInverterOn1 := FALSE;
            (* '<S1>:334:9' AMK_bInverterOn2=false; *)
            AMK_bInverterOn2 := FALSE;
            (* '<S1>:334:10' AMK_bInverterOn3=false; *)
            AMK_bInverterOn3 := FALSE;
            (* '<S1>:334:11' AMK_bInverterOn4=false; *)
            AMK_bInverterOn4 := FALSE;
            (* '<S1>:334:12' AMK_bEnable1=false; *)
            AMK_bEnable1 := FALSE;
            (* '<S1>:334:13' AMK_bEnable2=false; *)
            AMK_bEnable2 := FALSE;
            (* '<S1>:334:14' AMK_bEnable3=false; *)
            AMK_bEnable3 := FALSE;
            (* '<S1>:334:15' AMK_bEnable4=false; *)
            AMK_bEnable4 := FALSE;
            (* '<S1>:334:16' AMK_bDcOn1=false; *)
            AMK_bDcOn1 := FALSE;
            (* '<S1>:334:17' AMK_bDcOn2=false; *)
            AMK_bDcOn2 := FALSE;
            (* '<S1>:334:18' AMK_bDcOn3=false; *)
            AMK_bDcOn3 := FALSE;
            (* '<S1>:334:19' AMK_bDcOn4=false; *)
            AMK_bDcOn4 := FALSE;
            (* Entry 'ERROR_INVERTER': '<S1>:381' *)
            (* Entry Internal 'ERROR_INVERTER': '<S1>:381' *)
            (* Transition: '<S1>:387' *)
            is_ERROR_INVERTER := UPMRacing_14E_StateMachine_IN_NO_ERROR;
            (* Outport: '<Root>/Estado_Error' incorporates:
             *  Outport: '<Root>/AMK_TargetVelocity1'
             *  Outport: '<Root>/AMK_TargetVelocity2'
             *  Outport: '<Root>/AMK_TargetVelocity3'
             *  Outport: '<Root>/AMK_TargetVelocity4'
             *  Outport: '<Root>/AMK_TorqueLimitNegativ1'
             *  Outport: '<Root>/AMK_TorqueLimitNegativ2'
             *  Outport: '<Root>/AMK_TorqueLimitNegativ3'
             *  Outport: '<Root>/AMK_TorqueLimitNegativ4'
             *  Outport: '<Root>/AMK_TorqueLimitPositiv1'
             *  Outport: '<Root>/AMK_TorqueLimitPositiv2'
             *  Outport: '<Root>/AMK_TorqueLimitPositiv3'
             *  Outport: '<Root>/AMK_TorqueLimitPositiv4'
             *  Outport: '<Root>/AMK_bDcOn1'
             *  Outport: '<Root>/AMK_bDcOn2'
             *  Outport: '<Root>/AMK_bDcOn3'
             *  Outport: '<Root>/AMK_bDcOn4'
             *  Outport: '<Root>/AMK_bEnable1'
             *  Outport: '<Root>/AMK_bEnable2'
             *  Outport: '<Root>/AMK_bEnable3'
             *  Outport: '<Root>/AMK_bEnable4'
             *  Outport: '<Root>/AMK_bInverterOn1'
             *  Outport: '<Root>/AMK_bInverterOn2'
             *  Outport: '<Root>/AMK_bInverterOn3'
             *  Outport: '<Root>/AMK_bInverterOn4'
             *  Outport: '<Root>/Estado'
             *  Outport: '<Root>/Pre_Charge' *)
            (* Entry 'NO_ERROR': '<S1>:384' *)
            (* No hay errores *)
            (* '<S1>:384:3' Estado_Error = 11; *)
            Estado_Error := 11;
            (* Entry 'BRAKE_LIGHT': '<S1>:519' *)
            (* Entry Internal 'BRAKE_LIGHT': '<S1>:519' *)
            (* Transition: '<S1>:521' *)
            is_BRAKE_LIGHT := UPMRacing_14E_StateMachine_IN_LIGHT_OFF;
            (* Entry 'LIGHT_OFF': '<S1>:520' *)
            (* Entry 'COOLING_RIGHT': '<S1>:526' *)
            (* Entry Internal 'COOLING_RIGHT': '<S1>:526' *)
            (* Transition: '<S1>:610' *)
            is_COOLING_RIGHT := UPMRacing_14E_StateMachine_IN_COOLING_OFF_RIGHT;
            (* Entry 'COOLING_OFF_RIGHT': '<S1>:612' *)
            (* '<S1>:612:2' Cooling_Pumps_On = false; *)
            (* '<S1>:612:3' Fan_Left = false; *)
            (* Entry 'COOLING_LEFT': '<S1>:543' *)
            (* Entry Internal 'COOLING_LEFT': '<S1>:543' *)
            (* Transition: '<S1>:547' *)
            is_COOLING_LEFT := UPMRacing_14E_StateMachine_IN_COOLING_OFF_LEFT;
            (* Entry 'COOLING_OFF_LEFT': '<S1>:602' *)
            (* '<S1>:602:2' Cooling_Pumps_On = false; *)
            Cooling_Pumps_On := FALSE;
            (* '<S1>:602:3' Fan_Left = false; *)
            Fan_Left := FALSE;
        ELSE 
            (* During 'CAR': '<S1>:380' *)
            temp10 := FALSE;
            temp8 := FALSE;
            temp9 := FALSE;

            CASE is_CAR OF
                UPMRacing_14E_StateMachine_IN_DRIVE: 
                    (* During 'DRIVE': '<S1>:169' *)
                    (* '<S1>:815:1' sf_internal_predicateOutput = BMS_Voltage < BMS_Voltage_Min; *)

                    IF BMS_Voltage < BMS_Voltage_Min THEN 
                        (* Transition: '<S1>:815' *)
                        temp9 := TRUE;
                    ELSE 
                        (* '<S1>:932:1' sf_internal_predicateOutput = AccPedal_1<0 || AccPedal_1>5000; *)

                        IF AccPedal_1 > 5000 THEN 
                            sf_internal_predicateOutput := TRUE;
                        ELSE 
                            sf_internal_predicateOutput := FALSE;
                        END_IF;


                        IF (((sf_internal_predicateOutput OR (Shutdown_Circuit < 6000)) OR (Wake_Up < 6000)) OR (AccPedal_2 > 5000)) OR ((Brake_Pedal <= 0) OR (Brake_Pedal > 5000)) THEN 
                            (* Transition: '<S1>:932' *)
                            (* Transition: '<S1>:635' *)
                            (* Transition: '<S1>:206' *)
                            (* Transition: '<S1>:933' *)
                            (* Transition: '<S1>:934' *)
                            temp9 := TRUE;
                        ELSE 
                            (* '<S1>:635:1' sf_internal_predicateOutput = Shutdown_Circuit<6000; *)
                            (* '<S1>:206:1' sf_internal_predicateOutput = Wake_Up < 6000; *)
                            (* '<S1>:933:1' sf_internal_predicateOutput = AccPedal_2<0 || AccPedal_2>5000; *)
                            (* '<S1>:934:1' sf_internal_predicateOutput = Brake_Pedal<=0 || Brake_Pedal>5000; *)
                            (* '<S1>:169:4' [Throttle,Implausibility] = Throttle_Control(AccPedal_1,AccPedal_2); *)
                            (* Simulink Function 'Throttle_Control': '<S1>:484' *)
                            b_AccPedal_1 := AccPedal_1;
                            b_AccPedal_2 := AccPedal_2;
                            i0_Throttle_Control(ssMethodType := SS_OUTPUT, AccPedal_1 := b_AccPedal_1, AccPedal_2 := b_AccPedal_2);
                            temp11 := i0_Throttle_Control.Throttle;
                            sf_internal_predicateOutput := i0_Throttle_Control.Implausibility;
                            Compare_d := sf_internal_predicateOutput;
                            Saturation := temp11;
                            Throttle := Saturation;

                            CASE is_DRIVE OF
                                UPMRacing_14E_StateMachine_IN_Accelerate: 
                                    (* During 'Accelerate': '<S1>:146' *)
                                    (* State where the motors are active. It's allways an acceleration state. If acceleration is 0, then it wil keep constant velocity. *)
                                    (* '<S1>:438:1' sf_internal_predicateOutput = Inverter_Error == 1; *)

                                    IF Inverter_Error THEN 
                                        (* Transition: '<S1>:438' *)
                                        is_DRIVE := UPMRacing_14E_StateMachine_IN_Error_Drive;
                                        (* Entry 'Error_Drive': '<S1>:437' *)
                                        (* '<S1>:437:2' Estado = 23; *)
                                        Estado := 23;
                                        (* '<S1>:437:3' AMK_bEnable1=false; *)
                                        AMK_bEnable1 := FALSE;
                                        (* '<S1>:437:3' AMK_bEnable2=false; *)
                                        AMK_bEnable2 := FALSE;
                                        (* '<S1>:437:3' AMK_bEnable3=false; *)
                                        AMK_bEnable3 := FALSE;
                                        (* '<S1>:437:3' AMK_bEnable4=false; *)
                                        AMK_bEnable4 := FALSE;
                                        (* '<S1>:437:4' AMK_bInverterOn1=false; *)
                                        AMK_bInverterOn1 := FALSE;
                                        (* '<S1>:437:4' AMK_bInverterOn2=false; *)
                                        AMK_bInverterOn2 := FALSE;
                                        (* '<S1>:437:4' AMK_bInverterOn3=false; *)
                                        AMK_bInverterOn3 := FALSE;
                                        (* '<S1>:437:4' AMK_bInverterOn4=false; *)
                                        AMK_bInverterOn4 := FALSE;
                                        (* '<S1>:437:5' AMK_bDcOn1=false; *)
                                        AMK_bDcOn1 := FALSE;
                                        (* '<S1>:437:5' AMK_bDcOn2=false; *)
                                        AMK_bDcOn2 := FALSE;
                                        (* '<S1>:437:5' AMK_bDcOn3=false; *)
                                        AMK_bDcOn3 := FALSE;
                                        (* '<S1>:437:5' AMK_bDcOn4=false; *)
                                        AMK_bDcOn4 := FALSE;
                                    ELSE 
                                        (* '<S1>:560:1' sf_internal_predicateOutput = Throttle>=0.25 &amp; Brake_Pedal <= Braking_OffSet; *)

                                        IF (Saturation >= 0.25) AND (Brake_Pedal <= Braking_OffSet) THEN 
                                            (* Transition: '<S1>:560' *)
                                            is_DRIVE := UPMRacing_14E_StateMachine_IN_BRAKE_PLAUSIBILITY_CHECK;
                                            (* Entry 'BRAKE_PLAUSIBILITY_CHECK': '<S1>:559' *)
                                            (* '<S1>:559:2' Estado = 25; *)
                                            Estado := 25;
                                        ELSE 
                                            (* '<S1>:171:1' sf_internal_predicateOutput = Throttle<=0 || Brake_Pedal <= Braking_OffSet; *)

                                            IF (Saturation <= 0.0) OR (Brake_Pedal <= Braking_OffSet) THEN 
                                                (* Transition: '<S1>:171' *)
                                                is_DRIVE := UPMRacing_14E_StateMachine_IN_BRAKE;
                                                (* Entry 'BRAKE': '<S1>:170' *)
                                                (* '<S1>:170:2' Estado = 22; *)
                                                Estado := 22;
                                            ELSE 
                                                (* '<S1>:499:1' sf_internal_predicateOutput = Implausibility==true; *)

                                                IF Compare_d THEN 
                                                    (* Transition: '<S1>:499' *)
                                                    is_DRIVE := UPMRacing_14E_StateMachine_IN_IMPLAUSIBILITY_STATUS;
                                                    temporalCounter_i1(timerAction := 1, maxTime := 0);
                                                    (* Entry 'IMPLAUSIBILITY_STATUS': '<S1>:498' *)
                                                    (* '<S1>:498:2' Estado = 24; *)
                                                    Estado := 24;
                                                ELSE 
                                                    (* '<S1>:811:1' sf_internal_predicateOutput = Drive_Button < 12000; *)

                                                    IF Drive_Button < 12000 THEN 
                                                        (* Transition: '<S1>:811' *)
                                                        (* Transition: '<S1>:866' *)
                                                        is_DRIVE := UPMRacing_14E_StateMachine_IN_PRE_DRIVE;
                                                        (* Entry 'PRE_DRIVE': '<S1>:503' *)
                                                        (* '<S1>:503:2' Estado = 20; *)
                                                        Estado := 20;
                                                    ELSE 
                                                        (* '<S1>:866:1' sf_internal_predicateOutput = Drive_Button < 12000; *)
                                                        (* '<S1>:146:4' [AMK_TorqueLimitPositiv1,AMK_TorqueLimitPositiv2,AMK_TorqueLimitPositiv3,AMK_TorqueLimitPositiv4,... *)
                                                        (* '<S1>:146:5'        Speed_RPM,AMK_TorqueLimitNegativ1,AMK_TorqueLimitNegativ2,AMK_TorqueLimitNegativ3,AMK_TorqueLimitNegativ4,... *)
                                                        (* '<S1>:146:6'        AMK_TargetVelocity1,AMK_TargetVelocity2,AMK_TargetVelocity3,AMK_TargetVelocity4] = Yaw_Control(AMK_ActualVelocity1... *)
                                                        (* '<S1>:146:7'        ,AMK_ActualVelocity2,AMK_ActualVelocity3,AMK_ActualVelocity4,Throttle,Steering_Wheel_Angle,Yaw_Rate_AIM); *)
                                                        (* Simulink Function 'Yaw_Control': '<S1>:839' *)
                                                        b_AMK_ActualVelocity1 := AMK_ActualVelocity1;
                                                        b_AMK_ActualVelocity2 := AMK_ActualVelocity2;
                                                        b_AMK_ActualVelocity3 := AMK_ActualVelocity3;
                                                        b_AMK_ActualVelocity4 := AMK_ActualVelocity4;
                                                        Throttle_a := Saturation;
                                                        b_Steering_Wheel_Angle := Steering_Wheel_Angle;
                                                        b_Yaw_Rate_AIM := Yaw_Rate_AIM;
                                                        i0_Yaw_Control(ssMethodType := SS_OUTPUT, AMK_ActualVelocity1 := b_AMK_ActualVelocity1, AMK_ActualVelocity2 := b_AMK_ActualVelocity2, AMK_ActualVelocity3 := b_AMK_ActualVelocity3, AMK_ActualVelocity4 := b_AMK_ActualVelocity4, Throttle := Throttle_a, Steering_Wheel_Angle := b_Steering_Wheel_Angle, Yaw_Rate_AIM := b_Yaw_Rate_AIM);
                                                        temp12 := i0_Yaw_Control.AMK_TorqueLimitPositiv1;
                                                        temp13 := i0_Yaw_Control.AMK_TorqueLimitPositiv2;
                                                        temp14 := i0_Yaw_Control.AMK_TorqueLimitPositiv3;
                                                        temp15 := i0_Yaw_Control.AMK_TorqueLimitPositiv4;
                                                        temp16 := i0_Yaw_Control.Speed_RPM;
                                                        temp17 := i0_Yaw_Control.AMK_TorqueLimitNegativ1;
                                                        temp18 := i0_Yaw_Control.AMK_TorqueLimitNegativ2;
                                                        temp19 := i0_Yaw_Control.AMK_TorqueLimitNegativ3;
                                                        temp20 := i0_Yaw_Control.AMK_TorqueLimitNegativ4;
                                                        temp21 := i0_Yaw_Control.AMK_TargetVelocity1;
                                                        temp22 := i0_Yaw_Control.AMK_TargetVelocity2;
                                                        temp23 := i0_Yaw_Control.AMK_TargetVelocity3;
                                                        temp24 := i0_Yaw_Control.AMK_TargetVelocity4;
                                                        OutportBufferForAMK_TargetVelocity4 := temp24;
                                                        OutportBufferForAMK_TargetVelocity3 := temp23;
                                                        OutportBufferForAMK_TargetVelocity2 := temp22;
                                                        DataTypeConversion3 := temp21;
                                                        OutportBufferForAMK_TorqueLimitNegativ4 := temp20;
                                                        OutportBufferForAMK_TorqueLimitNegativ3 := temp19;
                                                        OutportBufferForAMK_TorqueLimitNegativ2 := temp18;
                                                        DataTypeConversion6 := temp17;
                                                        DataTypeConversion := temp16;
                                                        DataTypeConversion5 := temp15;
                                                        DataTypeConversion4 := temp14;
                                                        DataTypeConversion2 := temp13;
                                                        DataTypeConversion1 := temp12;
                                                        AMK_TorqueLimitPositiv1 := DataTypeConversion1;
                                                        AMK_TorqueLimitPositiv2 := DataTypeConversion2;
                                                        AMK_TorqueLimitPositiv3 := DataTypeConversion4;
                                                        AMK_TorqueLimitPositiv4 := DataTypeConversion5;
                                                        Speed_RPM := DataTypeConversion;
                                                        AMK_TorqueLimitNegativ1 := DataTypeConversion6;
                                                        AMK_TorqueLimitNegativ2 := OutportBufferForAMK_TorqueLimitNegativ2;
                                                        AMK_TorqueLimitNegativ3 := OutportBufferForAMK_TorqueLimitNegativ3;
                                                        AMK_TorqueLimitNegativ4 := OutportBufferForAMK_TorqueLimitNegativ4;
                                                        AMK_TargetVelocity1 := DataTypeConversion3;
                                                        AMK_TargetVelocity2 := OutportBufferForAMK_TargetVelocity2;
                                                        AMK_TargetVelocity3 := OutportBufferForAMK_TargetVelocity3;
                                                        AMK_TargetVelocity4 := OutportBufferForAMK_TargetVelocity4;
                                                    END_IF;

                                                END_IF;

                                            END_IF;

                                        END_IF;

                                    END_IF;

                                UPMRacing_14E_StateMachine_IN_BRAKE: 
                                    (* During 'BRAKE': '<S1>:170' *)
                                    (* '<S1>:511:1' sf_internal_predicateOutput = Inverter_Error == 1; *)

                                    IF Inverter_Error THEN 
                                        (* Transition: '<S1>:511' *)
                                        is_DRIVE := UPMRacing_14E_StateMachine_IN_Error_Drive;
                                        (* Entry 'Error_Drive': '<S1>:437' *)
                                        (* '<S1>:437:2' Estado = 23; *)
                                        Estado := 23;
                                        (* '<S1>:437:3' AMK_bEnable1=false; *)
                                        AMK_bEnable1 := FALSE;
                                        (* '<S1>:437:3' AMK_bEnable2=false; *)
                                        AMK_bEnable2 := FALSE;
                                        (* '<S1>:437:3' AMK_bEnable3=false; *)
                                        AMK_bEnable3 := FALSE;
                                        (* '<S1>:437:3' AMK_bEnable4=false; *)
                                        AMK_bEnable4 := FALSE;
                                        (* '<S1>:437:4' AMK_bInverterOn1=false; *)
                                        AMK_bInverterOn1 := FALSE;
                                        (* '<S1>:437:4' AMK_bInverterOn2=false; *)
                                        AMK_bInverterOn2 := FALSE;
                                        (* '<S1>:437:4' AMK_bInverterOn3=false; *)
                                        AMK_bInverterOn3 := FALSE;
                                        (* '<S1>:437:4' AMK_bInverterOn4=false; *)
                                        AMK_bInverterOn4 := FALSE;
                                        (* '<S1>:437:5' AMK_bDcOn1=false; *)
                                        AMK_bDcOn1 := FALSE;
                                        (* '<S1>:437:5' AMK_bDcOn2=false; *)
                                        AMK_bDcOn2 := FALSE;
                                        (* '<S1>:437:5' AMK_bDcOn3=false; *)
                                        AMK_bDcOn3 := FALSE;
                                        (* '<S1>:437:5' AMK_bDcOn4=false; *)
                                        AMK_bDcOn4 := FALSE;
                                    ELSE 
                                        (* '<S1>:172:1' sf_internal_predicateOutput = Throttle>0 &amp; Implausibility==false &amp; Brake_Pedal > Braking_OffSet; *)

                                        IF ((Saturation > 0.0) AND ( NOT Compare_d)) AND (Brake_Pedal > Braking_OffSet) THEN 
                                            (* Transition: '<S1>:172' *)
                                            is_DRIVE := UPMRacing_14E_StateMachine_IN_Accelerate;
                                            (* Entry 'Accelerate': '<S1>:146' *)
                                            (* '<S1>:146:2' Estado = 21; *)
                                            Estado := 21;
                                        ELSE 
                                            (* '<S1>:509:1' sf_internal_predicateOutput = Drive_Button < 12000; *)

                                            IF Drive_Button < 12000 THEN 
                                                (* Transition: '<S1>:509' *)
                                                is_DRIVE := UPMRacing_14E_StateMachine_IN_PRE_DRIVE;
                                                (* Entry 'PRE_DRIVE': '<S1>:503' *)
                                                (* '<S1>:503:2' Estado = 20; *)
                                                Estado := 20;
                                            ELSE 
                                                (* '<S1>:170:4' [AMK_TargetVelocity1, AMK_TargetVelocity2, AMK_TargetVelocity3, AMK_TargetVelocity4]=Constant(int16(20000)); *)
                                                (* Simulink Function 'Constant': '<S1>:190' *)
                                                x := 20000;
                                                i0_b_Constant(ssMethodType := SS_OUTPUT, x := x);
                                                temp12 := i0_b_Constant.y1;
                                                temp13 := i0_b_Constant.y2;
                                                temp14 := i0_b_Constant.y3;
                                                temp15 := i0_b_Constant.y4;
                                                OutportBufferFory4 := temp15;
                                                OutportBufferFory3 := temp14;
                                                OutportBufferFory2 := temp13;
                                                x_l := temp12;
                                                AMK_TargetVelocity1 := x_l;
                                                AMK_TargetVelocity2 := OutportBufferFory2;
                                                AMK_TargetVelocity3 := OutportBufferFory3;
                                                AMK_TargetVelocity4 := OutportBufferFory4;
                                                (* '<S1>:170:5' [AMK_TorqueLimitPositiv1, AMK_TorqueLimitPositiv2, AMK_TorqueLimitPositiv3, AMK_TorqueLimitPositiv4... *)
                                                (* '<S1>:170:6'       ]=Constant(int16(0)); *)
                                                (* Simulink Function 'Constant': '<S1>:190' *)
                                                x := 0;
                                                i0_b_Constant(ssMethodType := SS_OUTPUT, x := x);
                                                temp12 := i0_b_Constant.y1;
                                                temp13 := i0_b_Constant.y2;
                                                temp14 := i0_b_Constant.y3;
                                                temp15 := i0_b_Constant.y4;
                                                OutportBufferFory4 := temp15;
                                                OutportBufferFory3 := temp14;
                                                OutportBufferFory2 := temp13;
                                                x_l := temp12;
                                                AMK_TorqueLimitPositiv1 := x_l;
                                                AMK_TorqueLimitPositiv2 := OutportBufferFory2;
                                                AMK_TorqueLimitPositiv3 := OutportBufferFory3;
                                                AMK_TorqueLimitPositiv4 := OutportBufferFory4;
                                                (* '<S1>:170:7' [AMK_TorqueLimitNegativ1, AMK_TorqueLimitNegativ2, AMK_TorqueLimitNegativ3, AMK_TorqueLimitNegativ4... *)
                                                (* '<S1>:170:8'       ]=Constant(int16(0)); *)
                                                (* Simulink Function 'Constant': '<S1>:190' *)
                                                x := 0;
                                                i0_b_Constant(ssMethodType := SS_OUTPUT, x := x);
                                                temp12 := i0_b_Constant.y1;
                                                temp13 := i0_b_Constant.y2;
                                                temp14 := i0_b_Constant.y3;
                                                temp15 := i0_b_Constant.y4;
                                                OutportBufferFory4 := temp15;
                                                OutportBufferFory3 := temp14;
                                                OutportBufferFory2 := temp13;
                                                x_l := temp12;
                                                AMK_TorqueLimitNegativ1 := x_l;
                                                AMK_TorqueLimitNegativ2 := OutportBufferFory2;
                                                AMK_TorqueLimitNegativ3 := OutportBufferFory3;
                                                AMK_TorqueLimitNegativ4 := OutportBufferFory4;
                                            END_IF;

                                        END_IF;

                                    END_IF;

                                UPMRacing_14E_StateMachine_IN_BRAKE_PLAUSIBILITY_CHECK: 
                                    (* During 'BRAKE_PLAUSIBILITY_CHECK': '<S1>:559' *)
                                    (* '<S1>:562:1' sf_internal_predicateOutput = Throttle<0.05; *)

                                    IF REAL_TO_LREAL(Saturation) < 0.05 THEN 
                                        (* Transition: '<S1>:562' *)
                                        temp10 := TRUE;
                                    ELSE 
                                        (* '<S1>:563:1' sf_internal_predicateOutput = Throttle<=0 || Brake_Pedal <= Braking_OffSet; *)

                                        IF (Saturation <= 0.0) OR (Brake_Pedal <= Braking_OffSet) THEN 
                                            (* Transition: '<S1>:563' *)
                                            is_DRIVE := UPMRacing_14E_StateMachine_IN_BRAKE;
                                            (* Entry 'BRAKE': '<S1>:170' *)
                                            (* '<S1>:170:2' Estado = 22; *)
                                            Estado := 22;
                                        ELSE 
                                            (* '<S1>:812:1' sf_internal_predicateOutput = Drive_Button < 12000; *)

                                            IF Drive_Button < 12000 THEN 
                                                (* Transition: '<S1>:812' *)
                                                temp10 := TRUE;
                                            ELSE 
                                                (* '<S1>:559:4' [AMK_TargetVelocity1, AMK_TargetVelocity2, AMK_TargetVelocity3, AMK_TargetVelocity4]=Constant(int16(20000)); *)
                                                (* Simulink Function 'Constant': '<S1>:190' *)
                                                x := 20000;
                                                i0_b_Constant(ssMethodType := SS_OUTPUT, x := x);
                                                temp12 := i0_b_Constant.y1;
                                                temp13 := i0_b_Constant.y2;
                                                temp14 := i0_b_Constant.y3;
                                                temp15 := i0_b_Constant.y4;
                                                OutportBufferFory4 := temp15;
                                                OutportBufferFory3 := temp14;
                                                OutportBufferFory2 := temp13;
                                                x_l := temp12;
                                                AMK_TargetVelocity1 := x_l;
                                                AMK_TargetVelocity2 := OutportBufferFory2;
                                                AMK_TargetVelocity3 := OutportBufferFory3;
                                                AMK_TargetVelocity4 := OutportBufferFory4;
                                                (* '<S1>:559:5' [AMK_TorqueLimitPositiv1, AMK_TorqueLimitPositiv2, AMK_TorqueLimitPositiv3, AMK_TorqueLimitPositiv4... *)
                                                (* '<S1>:559:6'       ]=Constant(int16(0)); *)
                                                (* Simulink Function 'Constant': '<S1>:190' *)
                                                x := 0;
                                                i0_b_Constant(ssMethodType := SS_OUTPUT, x := x);
                                                temp12 := i0_b_Constant.y1;
                                                temp13 := i0_b_Constant.y2;
                                                temp14 := i0_b_Constant.y3;
                                                temp15 := i0_b_Constant.y4;
                                                OutportBufferFory4 := temp15;
                                                OutportBufferFory3 := temp14;
                                                OutportBufferFory2 := temp13;
                                                x_l := temp12;
                                                AMK_TorqueLimitPositiv1 := x_l;
                                                AMK_TorqueLimitPositiv2 := OutportBufferFory2;
                                                AMK_TorqueLimitPositiv3 := OutportBufferFory3;
                                                AMK_TorqueLimitPositiv4 := OutportBufferFory4;
                                                (* '<S1>:559:7' [AMK_TorqueLimitNegativ1, AMK_TorqueLimitNegativ2, AMK_TorqueLimitNegativ3, AMK_TorqueLimitNegativ4... *)
                                                (* '<S1>:559:8'       ]=Constant(int16(0)); *)
                                                (* Simulink Function 'Constant': '<S1>:190' *)
                                                x := 0;
                                                i0_b_Constant(ssMethodType := SS_OUTPUT, x := x);
                                                temp12 := i0_b_Constant.y1;
                                                temp13 := i0_b_Constant.y2;
                                                temp14 := i0_b_Constant.y3;
                                                temp15 := i0_b_Constant.y4;
                                                OutportBufferFory4 := temp15;
                                                OutportBufferFory3 := temp14;
                                                OutportBufferFory2 := temp13;
                                                x_l := temp12;
                                                AMK_TorqueLimitNegativ1 := x_l;
                                                AMK_TorqueLimitNegativ2 := OutportBufferFory2;
                                                AMK_TorqueLimitNegativ3 := OutportBufferFory3;
                                                AMK_TorqueLimitNegativ4 := OutportBufferFory4;
                                            END_IF;

                                        END_IF;

                                    END_IF;

                                UPMRacing_14E_StateMachine_IN_Error_Drive: 
                                    (* During 'Error_Drive': '<S1>:437' *)
                                    (* '<S1>:439:1' sf_internal_predicateOutput = Inverter_Error == 0 &amp; Wake_Up > 6000; *)

                                    IF ( NOT Inverter_Error) AND (Wake_Up > 6000) THEN 
                                        (* Transition: '<S1>:439' *)
                                        is_DRIVE := UPMRacing_14E_StateMachine_IN_NO_ACTIVE_CHILD;
                                        is_CAR := UPMRacing_14E_StateMachine_IN_POWER_MOTOR_ON;
                                        (* Entry 'POWER_MOTOR_ON': '<S1>:137' *)
                                        (* '<S1>:137:2' Cooling_Enable = true; *)
                                        Cooling_Enable := TRUE;
                                        (* Entry Internal 'POWER_MOTOR_ON': '<S1>:137' *)
                                        (* Transition: '<S1>:210' *)
                                        is_POWER_MOTOR_ON := UPMRacing_14E_StateMachine_IN_INVERTER_ON;
                                        (* Entry 'INVERTER_ON': '<S1>:163' *)
                                        (* '<S1>:163:3' Estado = 11; *)
                                        Estado := 11;
                                    ELSE 
                                        (* '<S1>:437:7' [AMK_TargetVelocity1, AMK_TargetVelocity2, AMK_TargetVelocity3, AMK_TargetVelocity4]=Constant(int16(0)); *)
                                        (* Simulink Function 'Constant': '<S1>:190' *)
                                        x := 0;
                                        i0_b_Constant(ssMethodType := SS_OUTPUT, x := x);
                                        temp12 := i0_b_Constant.y1;
                                        temp13 := i0_b_Constant.y2;
                                        temp14 := i0_b_Constant.y3;
                                        temp15 := i0_b_Constant.y4;
                                        OutportBufferFory4 := temp15;
                                        OutportBufferFory3 := temp14;
                                        OutportBufferFory2 := temp13;
                                        x_l := temp12;
                                        AMK_TargetVelocity1 := x_l;
                                        AMK_TargetVelocity2 := OutportBufferFory2;
                                        AMK_TargetVelocity3 := OutportBufferFory3;
                                        AMK_TargetVelocity4 := OutportBufferFory4;
                                        (* '<S1>:437:8' [AMK_TorqueLimitPositiv1, AMK_TorqueLimitPositiv2, AMK_TorqueLimitPositiv3, AMK_TorqueLimitPositiv4... *)
                                        (* '<S1>:437:9'     ]=Constant(int16(0)); *)
                                        (* Simulink Function 'Constant': '<S1>:190' *)
                                        x := 0;
                                        i0_b_Constant(ssMethodType := SS_OUTPUT, x := x);
                                        temp12 := i0_b_Constant.y1;
                                        temp13 := i0_b_Constant.y2;
                                        temp14 := i0_b_Constant.y3;
                                        temp15 := i0_b_Constant.y4;
                                        OutportBufferFory4 := temp15;
                                        OutportBufferFory3 := temp14;
                                        OutportBufferFory2 := temp13;
                                        x_l := temp12;
                                        AMK_TorqueLimitPositiv1 := x_l;
                                        AMK_TorqueLimitPositiv2 := OutportBufferFory2;
                                        AMK_TorqueLimitPositiv3 := OutportBufferFory3;
                                        AMK_TorqueLimitPositiv4 := OutportBufferFory4;
                                        (* '<S1>:437:10' [AMK_TorqueLimitNegativ1, AMK_TorqueLimitNegativ2, AMK_TorqueLimitNegativ3, AMK_TorqueLimitNegativ4... *)
                                        (* '<S1>:437:11'     ]=Constant(int16(0)); *)
                                        (* Simulink Function 'Constant': '<S1>:190' *)
                                        x := 0;
                                        i0_b_Constant(ssMethodType := SS_OUTPUT, x := x);
                                        temp12 := i0_b_Constant.y1;
                                        temp13 := i0_b_Constant.y2;
                                        temp14 := i0_b_Constant.y3;
                                        temp15 := i0_b_Constant.y4;
                                        OutportBufferFory4 := temp15;
                                        OutportBufferFory3 := temp14;
                                        OutportBufferFory2 := temp13;
                                        x_l := temp12;
                                        AMK_TorqueLimitNegativ1 := x_l;
                                        AMK_TorqueLimitNegativ2 := OutportBufferFory2;
                                        AMK_TorqueLimitNegativ3 := OutportBufferFory3;
                                        AMK_TorqueLimitNegativ4 := OutportBufferFory4;
                                    END_IF;

                                UPMRacing_14E_StateMachine_IN_IMPLAUSIBILITY_STATUS: 
                                    (* During 'IMPLAUSIBILITY_STATUS': '<S1>:498' *)
                                    (* '<S1>:500:1' sf_internal_predicateOutput = Implausibility==false; *)

                                    IF  NOT Compare_d THEN 
                                        (* Transition: '<S1>:500' *)
                                        is_DRIVE := UPMRacing_14E_StateMachine_IN_Accelerate;
                                        (* Entry 'Accelerate': '<S1>:146' *)
                                        (* '<S1>:146:2' Estado = 21; *)
                                        Estado := 21;
                                    ELSE 
                                        (* '<S1>:502:1' sf_internal_predicateOutput = Throttle<=0 || Brake_Pedal <= Braking_OffSet; *)

                                        IF (Saturation <= 0.0) OR (Brake_Pedal <= Braking_OffSet) THEN 
                                            (* Transition: '<S1>:502' *)
                                            temp8 := TRUE;
                                        ELSE 
                                            (* '<S1>:501:1' sf_internal_predicateOutput = after(70,msec); *)
                                            temporalCounter_i1(timerAction := 2, maxTime := 70);

                                            IF temporalCounter_i1.done THEN 
                                                (* Transition: '<S1>:501' *)
                                                temp8 := TRUE;
                                            ELSE 
                                                (* '<S1>:498:4' [AMK_TorqueLimitPositiv1,AMK_TorqueLimitPositiv2,AMK_TorqueLimitPositiv3,AMK_TorqueLimitPositiv4,... *)
                                                (* '<S1>:498:5'     Speed_RPM,AMK_TorqueLimitNegativ1,AMK_TorqueLimitNegativ2,AMK_TorqueLimitNegativ3,... *)
                                                (* '<S1>:498:6'     AMK_TorqueLimitNegativ4,AMK_TargetVelocity1,AMK_TargetVelocity2,AMK_TargetVelocity3,... *)
                                                (* '<S1>:498:7'     AMK_TargetVelocity4] = Yaw_Control(AMK_ActualVelocity1,AMK_ActualVelocity2,AMK_ActualVelocity3,... *)
                                                (* '<S1>:498:8'     AMK_ActualVelocity4,Throttle,Steering_Wheel_Angle,Yaw_Rate_AIM); *)
                                                (* Simulink Function 'Yaw_Control': '<S1>:839' *)
                                                b_AMK_ActualVelocity1 := AMK_ActualVelocity1;
                                                b_AMK_ActualVelocity2 := AMK_ActualVelocity2;
                                                b_AMK_ActualVelocity3 := AMK_ActualVelocity3;
                                                b_AMK_ActualVelocity4 := AMK_ActualVelocity4;
                                                Throttle_a := Throttle;
                                                b_Steering_Wheel_Angle := Steering_Wheel_Angle;
                                                b_Yaw_Rate_AIM := Yaw_Rate_AIM;
                                                i0_Yaw_Control(ssMethodType := SS_OUTPUT, AMK_ActualVelocity1 := b_AMK_ActualVelocity1, AMK_ActualVelocity2 := b_AMK_ActualVelocity2, AMK_ActualVelocity3 := b_AMK_ActualVelocity3, AMK_ActualVelocity4 := b_AMK_ActualVelocity4, Throttle := Throttle_a, Steering_Wheel_Angle := b_Steering_Wheel_Angle, Yaw_Rate_AIM := b_Yaw_Rate_AIM);
                                                temp12 := i0_Yaw_Control.AMK_TorqueLimitPositiv1;
                                                temp13 := i0_Yaw_Control.AMK_TorqueLimitPositiv2;
                                                temp14 := i0_Yaw_Control.AMK_TorqueLimitPositiv3;
                                                temp15 := i0_Yaw_Control.AMK_TorqueLimitPositiv4;
                                                temp16 := i0_Yaw_Control.Speed_RPM;
                                                temp17 := i0_Yaw_Control.AMK_TorqueLimitNegativ1;
                                                temp18 := i0_Yaw_Control.AMK_TorqueLimitNegativ2;
                                                temp19 := i0_Yaw_Control.AMK_TorqueLimitNegativ3;
                                                temp20 := i0_Yaw_Control.AMK_TorqueLimitNegativ4;
                                                temp21 := i0_Yaw_Control.AMK_TargetVelocity1;
                                                temp22 := i0_Yaw_Control.AMK_TargetVelocity2;
                                                temp23 := i0_Yaw_Control.AMK_TargetVelocity3;
                                                temp24 := i0_Yaw_Control.AMK_TargetVelocity4;
                                                OutportBufferForAMK_TargetVelocity4 := temp24;
                                                OutportBufferForAMK_TargetVelocity3 := temp23;
                                                OutportBufferForAMK_TargetVelocity2 := temp22;
                                                DataTypeConversion3 := temp21;
                                                OutportBufferForAMK_TorqueLimitNegativ4 := temp20;
                                                OutportBufferForAMK_TorqueLimitNegativ3 := temp19;
                                                OutportBufferForAMK_TorqueLimitNegativ2 := temp18;
                                                DataTypeConversion6 := temp17;
                                                DataTypeConversion := temp16;
                                                DataTypeConversion5 := temp15;
                                                DataTypeConversion4 := temp14;
                                                DataTypeConversion2 := temp13;
                                                DataTypeConversion1 := temp12;
                                                AMK_TorqueLimitPositiv1 := DataTypeConversion1;
                                                AMK_TorqueLimitPositiv2 := DataTypeConversion2;
                                                AMK_TorqueLimitPositiv3 := DataTypeConversion4;
                                                AMK_TorqueLimitPositiv4 := DataTypeConversion5;
                                                Speed_RPM := DataTypeConversion;
                                                AMK_TorqueLimitNegativ1 := DataTypeConversion6;
                                                AMK_TorqueLimitNegativ2 := OutportBufferForAMK_TorqueLimitNegativ2;
                                                AMK_TorqueLimitNegativ3 := OutportBufferForAMK_TorqueLimitNegativ3;
                                                AMK_TorqueLimitNegativ4 := OutportBufferForAMK_TorqueLimitNegativ4;
                                                AMK_TargetVelocity1 := DataTypeConversion3;
                                                AMK_TargetVelocity2 := OutportBufferForAMK_TargetVelocity2;
                                                AMK_TargetVelocity3 := OutportBufferForAMK_TargetVelocity3;
                                                AMK_TargetVelocity4 := OutportBufferForAMK_TargetVelocity4;
                                            END_IF;

                                        END_IF;

                                    END_IF;

                                UPMRacing_14E_StateMachine_IN_PRE_DRIVE: 
                                    (* During 'PRE_DRIVE': '<S1>:503' *)
                                    (* '<S1>:508:1' sf_internal_predicateOutput = Drive_Button > 12000 &amp; Brake_Pedal <= Braking_OffSet; *)

                                    IF (Drive_Button > 12000) AND (Brake_Pedal <= Braking_OffSet) THEN 
                                        (* Transition: '<S1>:508' *)
                                        is_DRIVE := UPMRacing_14E_StateMachine_IN_RTDS;
                                        temporalCounter_i1(timerAction := 1, maxTime := 0);
                                        (* Entry 'RTDS': '<S1>:555' *)
                                    ELSE 
                                        (* '<S1>:512:1' sf_internal_predicateOutput = Inverter_Error == 1; *)

                                        IF Inverter_Error THEN 
                                            (* Transition: '<S1>:512' *)
                                            is_DRIVE := UPMRacing_14E_StateMachine_IN_Error_Drive;
                                            (* Entry 'Error_Drive': '<S1>:437' *)
                                            (* '<S1>:437:2' Estado = 23; *)
                                            Estado := 23;
                                            (* '<S1>:437:3' AMK_bEnable1=false; *)
                                            AMK_bEnable1 := FALSE;
                                            (* '<S1>:437:3' AMK_bEnable2=false; *)
                                            AMK_bEnable2 := FALSE;
                                            (* '<S1>:437:3' AMK_bEnable3=false; *)
                                            AMK_bEnable3 := FALSE;
                                            (* '<S1>:437:3' AMK_bEnable4=false; *)
                                            AMK_bEnable4 := FALSE;
                                            (* '<S1>:437:4' AMK_bInverterOn1=false; *)
                                            AMK_bInverterOn1 := FALSE;
                                            (* '<S1>:437:4' AMK_bInverterOn2=false; *)
                                            AMK_bInverterOn2 := FALSE;
                                            (* '<S1>:437:4' AMK_bInverterOn3=false; *)
                                            AMK_bInverterOn3 := FALSE;
                                            (* '<S1>:437:4' AMK_bInverterOn4=false; *)
                                            AMK_bInverterOn4 := FALSE;
                                            (* '<S1>:437:5' AMK_bDcOn1=false; *)
                                            AMK_bDcOn1 := FALSE;
                                            (* '<S1>:437:5' AMK_bDcOn2=false; *)
                                            AMK_bDcOn2 := FALSE;
                                            (* '<S1>:437:5' AMK_bDcOn3=false; *)
                                            AMK_bDcOn3 := FALSE;
                                            (* '<S1>:437:5' AMK_bDcOn4=false; *)
                                            AMK_bDcOn4 := FALSE;
                                        ELSE 
                                            (* '<S1>:503:4' [AMK_TargetVelocity1, AMK_TargetVelocity2, AMK_TargetVelocity3, AMK_TargetVelocity4]=Constant(int16(0)); *)
                                            (* Simulink Function 'Constant': '<S1>:190' *)
                                            x := 0;
                                            i0_b_Constant(ssMethodType := SS_OUTPUT, x := x);
                                            temp12 := i0_b_Constant.y1;
                                            temp13 := i0_b_Constant.y2;
                                            temp14 := i0_b_Constant.y3;
                                            temp15 := i0_b_Constant.y4;
                                            OutportBufferFory4 := temp15;
                                            OutportBufferFory3 := temp14;
                                            OutportBufferFory2 := temp13;
                                            x_l := temp12;
                                            AMK_TargetVelocity1 := x_l;
                                            AMK_TargetVelocity2 := OutportBufferFory2;
                                            AMK_TargetVelocity3 := OutportBufferFory3;
                                            AMK_TargetVelocity4 := OutportBufferFory4;
                                            (* '<S1>:503:5' [AMK_TorqueLimitPositiv1, AMK_TorqueLimitPositiv2, AMK_TorqueLimitPositiv3, AMK_TorqueLimitPositiv4... *)
                                            (* '<S1>:503:6'       ]=Constant(int16(0)); *)
                                            (* Simulink Function 'Constant': '<S1>:190' *)
                                            x := 0;
                                            i0_b_Constant(ssMethodType := SS_OUTPUT, x := x);
                                            temp12 := i0_b_Constant.y1;
                                            temp13 := i0_b_Constant.y2;
                                            temp14 := i0_b_Constant.y3;
                                            temp15 := i0_b_Constant.y4;
                                            OutportBufferFory4 := temp15;
                                            OutportBufferFory3 := temp14;
                                            OutportBufferFory2 := temp13;
                                            x_l := temp12;
                                            AMK_TorqueLimitPositiv1 := x_l;
                                            AMK_TorqueLimitPositiv2 := OutportBufferFory2;
                                            AMK_TorqueLimitPositiv3 := OutportBufferFory3;
                                            AMK_TorqueLimitPositiv4 := OutportBufferFory4;
                                            (* '<S1>:503:7' [AMK_TorqueLimitNegativ1, AMK_TorqueLimitNegativ2, AMK_TorqueLimitNegativ3, AMK_TorqueLimitNegativ4... *)
                                            (* '<S1>:503:8'       ]=Constant(int16(0)); *)
                                            (* Simulink Function 'Constant': '<S1>:190' *)
                                            x := 0;
                                            i0_b_Constant(ssMethodType := SS_OUTPUT, x := x);
                                            temp12 := i0_b_Constant.y1;
                                            temp13 := i0_b_Constant.y2;
                                            temp14 := i0_b_Constant.y3;
                                            temp15 := i0_b_Constant.y4;
                                            OutportBufferFory4 := temp15;
                                            OutportBufferFory3 := temp14;
                                            OutportBufferFory2 := temp13;
                                            x_l := temp12;
                                            AMK_TorqueLimitNegativ1 := x_l;
                                            AMK_TorqueLimitNegativ2 := OutportBufferFory2;
                                            AMK_TorqueLimitNegativ3 := OutportBufferFory3;
                                            AMK_TorqueLimitNegativ4 := OutportBufferFory4;
                                        END_IF;

                                    END_IF;

                                ELSE
                                    (* During 'RTDS': '<S1>:555' *)
                                    (* '<S1>:557:1' sf_internal_predicateOutput = after(2,sec); *)
                                    temporalCounter_i1(timerAction := 2, maxTime := 2000);

                                    IF temporalCounter_i1.done THEN 
                                        (* Transition: '<S1>:557' *)
                                        (* Exit 'RTDS': '<S1>:555' *)
                                        (* '<S1>:555:8' RTDS_Sound = false; *)
                                        RTDS_Sound := FALSE;
                                        is_DRIVE := UPMRacing_14E_StateMachine_IN_BRAKE;
                                        (* Entry 'BRAKE': '<S1>:170' *)
                                        (* '<S1>:170:2' Estado = 22; *)
                                        Estado := 22;
                                    ELSE 
                                        (* '<S1>:556:1' sf_internal_predicateOutput = (Drive_Button < 12000) || ... *)
                                        (* '<S1>:556:2' Brake_Pedal > Braking_OffSet; *)

                                        IF (Drive_Button < 12000) OR (Brake_Pedal > Braking_OffSet) THEN 
                                            (* Transition: '<S1>:556' *)
                                            (* Exit 'RTDS': '<S1>:555' *)
                                            (* '<S1>:555:8' RTDS_Sound = false; *)
                                            RTDS_Sound := FALSE;
                                            is_DRIVE := UPMRacing_14E_StateMachine_IN_PRE_DRIVE;
                                            (* Entry 'PRE_DRIVE': '<S1>:503' *)
                                            (* '<S1>:503:2' Estado = 20; *)
                                            Estado := 20;
                                        ELSE 
                                            (* '<S1>:555:2' RTDS_Sound=true; *)
                                            RTDS_Sound := TRUE;
                                            (* '<S1>:555:3' [AMK_TargetVelocity1, AMK_TargetVelocity2, AMK_TargetVelocity3, AMK_TargetVelocity4]=Constant(int16(0)); *)
                                            (* Simulink Function 'Constant': '<S1>:190' *)
                                            x := 0;
                                            i0_b_Constant(ssMethodType := SS_OUTPUT, x := x);
                                            temp12 := i0_b_Constant.y1;
                                            temp13 := i0_b_Constant.y2;
                                            temp14 := i0_b_Constant.y3;
                                            temp15 := i0_b_Constant.y4;
                                            OutportBufferFory4 := temp15;
                                            OutportBufferFory3 := temp14;
                                            OutportBufferFory2 := temp13;
                                            x_l := temp12;
                                            AMK_TargetVelocity1 := x_l;
                                            AMK_TargetVelocity2 := OutportBufferFory2;
                                            AMK_TargetVelocity3 := OutportBufferFory3;
                                            AMK_TargetVelocity4 := OutportBufferFory4;
                                            (* '<S1>:555:4' [AMK_TorqueLimitPositiv1, AMK_TorqueLimitPositiv2, AMK_TorqueLimitPositiv3, AMK_TorqueLimitPositiv4... *)
                                            (* '<S1>:555:5'      ]=Constant(int16(0)); *)
                                            (* Simulink Function 'Constant': '<S1>:190' *)
                                            x := 0;
                                            i0_b_Constant(ssMethodType := SS_OUTPUT, x := x);
                                            temp12 := i0_b_Constant.y1;
                                            temp13 := i0_b_Constant.y2;
                                            temp14 := i0_b_Constant.y3;
                                            temp15 := i0_b_Constant.y4;
                                            OutportBufferFory4 := temp15;
                                            OutportBufferFory3 := temp14;
                                            OutportBufferFory2 := temp13;
                                            x_l := temp12;
                                            AMK_TorqueLimitPositiv1 := x_l;
                                            AMK_TorqueLimitPositiv2 := OutportBufferFory2;
                                            AMK_TorqueLimitPositiv3 := OutportBufferFory3;
                                            AMK_TorqueLimitPositiv4 := OutportBufferFory4;
                                            (* '<S1>:555:6' [AMK_TorqueLimitNegativ1, AMK_TorqueLimitNegativ2, AMK_TorqueLimitNegativ3, AMK_TorqueLimitNegativ4... *)
                                            (* '<S1>:555:7'      ]=Constant(int16(0)); *)
                                            (* Simulink Function 'Constant': '<S1>:190' *)
                                            x := 0;
                                            i0_b_Constant(ssMethodType := SS_OUTPUT, x := x);
                                            temp12 := i0_b_Constant.y1;
                                            temp13 := i0_b_Constant.y2;
                                            temp14 := i0_b_Constant.y3;
                                            temp15 := i0_b_Constant.y4;
                                            OutportBufferFory4 := temp15;
                                            OutportBufferFory3 := temp14;
                                            OutportBufferFory2 := temp13;
                                            x_l := temp12;
                                            AMK_TorqueLimitNegativ1 := x_l;
                                            AMK_TorqueLimitNegativ2 := OutportBufferFory2;
                                            AMK_TorqueLimitNegativ3 := OutportBufferFory3;
                                            AMK_TorqueLimitNegativ4 := OutportBufferFory4;
                                        END_IF;

                                    END_IF;

                            END_CASE;

                        END_IF;

                    END_IF;

                UPMRacing_14E_StateMachine_IN_IDLE: 
                    (* During 'IDLE': '<S1>:333' *)
                    (* '<S1>:333:11' [Throttle,Implausibility] = Throttle_Control(AccPedal_1,AccPedal_2); *)
                    (* Simulink Function 'Throttle_Control': '<S1>:484' *)
                    b_AccPedal_1 := AccPedal_1;
                    b_AccPedal_2 := AccPedal_2;
                    i0_Throttle_Control(ssMethodType := SS_OUTPUT, AccPedal_1 := b_AccPedal_1, AccPedal_2 := b_AccPedal_2);
                    temp11 := i0_Throttle_Control.Throttle;
                    sf_internal_predicateOutput := i0_Throttle_Control.Implausibility;
                    Compare_d := sf_internal_predicateOutput;
                    Saturation := temp11;
                    Throttle := Saturation;

                    CASE is_IDLE OF
                        UPMRacing_14E_StateMachine_IN_ERROR_PRECHARGE: 
                            (* During 'ERROR_PRECHARGE': '<S1>:617' *)
                            (* '<S1>:618:1' sf_internal_predicateOutput = Wake_Up < 6000; *)

                            IF Wake_Up < 6000 THEN 
                                (* Transition: '<S1>:618' *)
                                is_IDLE := UPMRacing_14E_StateMachine_IN_LVMS_ON;
                                (* Entry 'LVMS_ON': '<S1>:334' *)
                                (* In this state the ECU is waiting to start the inizialization of the inverters *)
                                (* Right now all LV systems are starting to initialize *)
                                (* '<S1>:334:4' Estado = 1; *)
                                Estado := 1;
                                (* Battery relays *)
                                (* '<S1>:334:6' Pre_Charge = false; *)
                                Pre_Charge := FALSE;
                                (* Inverters shutdown *)
                                (* '<S1>:334:8' AMK_bInverterOn1=false; *)
                                AMK_bInverterOn1 := FALSE;
                                (* '<S1>:334:9' AMK_bInverterOn2=false; *)
                                AMK_bInverterOn2 := FALSE;
                                (* '<S1>:334:10' AMK_bInverterOn3=false; *)
                                AMK_bInverterOn3 := FALSE;
                                (* '<S1>:334:11' AMK_bInverterOn4=false; *)
                                AMK_bInverterOn4 := FALSE;
                                (* '<S1>:334:12' AMK_bEnable1=false; *)
                                AMK_bEnable1 := FALSE;
                                (* '<S1>:334:13' AMK_bEnable2=false; *)
                                AMK_bEnable2 := FALSE;
                                (* '<S1>:334:14' AMK_bEnable3=false; *)
                                AMK_bEnable3 := FALSE;
                                (* '<S1>:334:15' AMK_bEnable4=false; *)
                                AMK_bEnable4 := FALSE;
                                (* '<S1>:334:16' AMK_bDcOn1=false; *)
                                AMK_bDcOn1 := FALSE;
                                (* '<S1>:334:17' AMK_bDcOn2=false; *)
                                AMK_bDcOn2 := FALSE;
                                (* '<S1>:334:18' AMK_bDcOn3=false; *)
                                AMK_bDcOn3 := FALSE;
                                (* '<S1>:334:19' AMK_bDcOn4=false; *)
                                AMK_bDcOn4 := FALSE;
                            END_IF;

                        ELSE
                            (* During 'LVMS_ON': '<S1>:334' *)
                            (* '<S1>:338:1' sf_internal_predicateOutput = (Wake_Up > 6000) &amp; ... *)
                            (* '<S1>:338:2' (BMS_Voltage > BMS_Voltage_Min); *)

                            IF (Wake_Up > 6000) AND (BMS_Voltage > BMS_Voltage_Min) THEN 
                                (* Transition: '<S1>:338' *)
                                is_IDLE := UPMRacing_14E_StateMachine_IN_NO_ACTIVE_CHILD;
                                (* Exit 'IDLE': '<S1>:333' *)
                                (* '<S1>:333:12' Throttle = single(0); *)
                                Throttle := 0.0;
                                (* '<S1>:333:12' Implausibility = false; *)
                                is_CAR := UPMRacing_14E_StateMachine_IN_POWER_MOTOR_ON;
                                (* Entry 'POWER_MOTOR_ON': '<S1>:137' *)
                                (* '<S1>:137:2' Cooling_Enable = true; *)
                                Cooling_Enable := TRUE;
                                (* Entry Internal 'POWER_MOTOR_ON': '<S1>:137' *)
                                (* Transition: '<S1>:210' *)
                                is_POWER_MOTOR_ON := UPMRacing_14E_StateMachine_IN_INVERTER_ON;
                                (* Entry 'INVERTER_ON': '<S1>:163' *)
                                (* '<S1>:163:3' Estado = 11; *)
                                Estado := 11;
                            END_IF;

                    END_CASE;

                UPMRacing_14E_StateMachine_IN_POWER_MOTOR_ON: 
                    (* During 'POWER_MOTOR_ON': '<S1>:137' *)
                    (* '<S1>:358:1' sf_internal_predicateOutput = Wake_Up < 6000; *)

